REGION Network 15: Interface Signals 10 BK8
   // Call the interface signals bool blocks
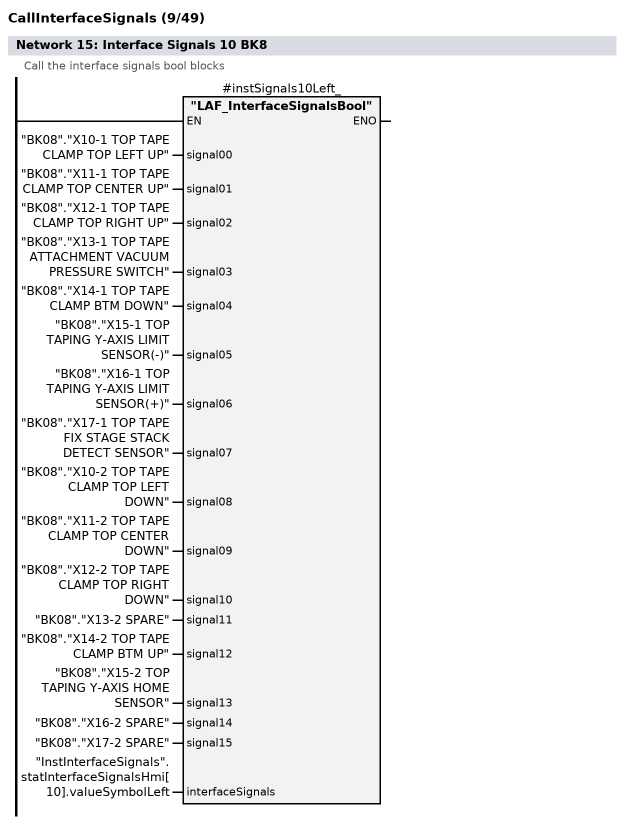
   RUNG wire#powerrail
      #instSignals10Left_(signal00 := "BK08"."X10-1 TOP TAPE CLAMP TOP LEFT UP", signal01 := "BK08"."X11-1 TOP TAPE CLAMP TOP CENTER UP", signal02 := "BK08"."X12-1 TOP TAPE CLAMP TOP RIGHT UP", signal03 := "BK08"."X13-1 TOP TAPE ATTACHMENT VACUUM PRESSURE SWITCH", signal04 := "BK08"."X14-1 TOP TAPE CLAMP BTM DOWN", signal05 := "BK08"."X15-1 TOP TAPING Y-AXIS LIMIT SENSOR(-)", signal06 := "BK08"."X16-1 TOP TAPING Y-AXIS LIMIT SENSOR(+)", signal07 := "BK08"."X17-1 TOP TAPE FIX STAGE STACK DETECT SENSOR", signal08 := "BK08"."X10-2 TOP TAPE CLAMP TOP LEFT DOWN", signal09 := "BK08"."X11-2 TOP TAPE CLAMP TOP CENTER DOWN", signal10 := "BK08"."X12-2 TOP TAPE CLAMP TOP RIGHT DOWN", signal11 := "BK08"."X13-2 SPARE", signal12 := "BK08"."X14-2 TOP TAPE CLAMP BTM UP", signal13 := "BK08"."X15-2 TOP TAPING Y-AXIS HOME SENSOR", signal14 := "BK08"."X16-2 SPARE", signal15 := "BK08"."X17-2 SPARE", interfaceSignals := "InstInterfaceSignals".statInterfaceSignalsHmi[10].valueSymbolLeft)
   END_RUNG
   // the same network as SCL:
   #instSignals10Left_(signal00 := "BK08"."X10-1 TOP TAPE CLAMP TOP LEFT UP",   // "LAF_InterfaceSignalsBool"
                       signal01 := "BK08"."X11-1 TOP TAPE CLAMP TOP CENTER UP",
                       signal02 := "BK08"."X12-1 TOP TAPE CLAMP TOP RIGHT UP",
                       signal03 := "BK08"."X13-1 TOP TAPE ATTACHMENT VACUUM PRESSURE SWITCH",
                       signal04 := "BK08"."X14-1 TOP TAPE CLAMP BTM DOWN",
                       signal05 := "BK08"."X15-1 TOP TAPING Y-AXIS LIMIT SENSOR(-)",
                       signal06 := "BK08"."X16-1 TOP TAPING Y-AXIS LIMIT SENSOR(+)",
                       signal07 := "BK08"."X17-1 TOP TAPE FIX STAGE STACK DETECT SENSOR",
                       signal08 := "BK08"."X10-2 TOP TAPE CLAMP TOP LEFT DOWN",
                       signal09 := "BK08"."X11-2 TOP TAPE CLAMP TOP CENTER DOWN",
                       signal10 := "BK08"."X12-2 TOP TAPE CLAMP TOP RIGHT DOWN",
                       signal11 := "BK08"."X13-2 SPARE",
                       signal12 := "BK08"."X14-2 TOP TAPE CLAMP BTM UP",
                       signal13 := "BK08"."X15-2 TOP TAPING Y-AXIS HOME SENSOR",
                       signal14 := "BK08"."X16-2 SPARE",
                       signal15 := "BK08"."X17-2 SPARE",
                       interfaceSignals := "InstInterfaceSignals".statInterfaceSignalsHmi[10].valueSymbolLeft);
END_REGION

REGION Network 16: Interface Signals 11 BK9
   // Call the interface signals bool blocks
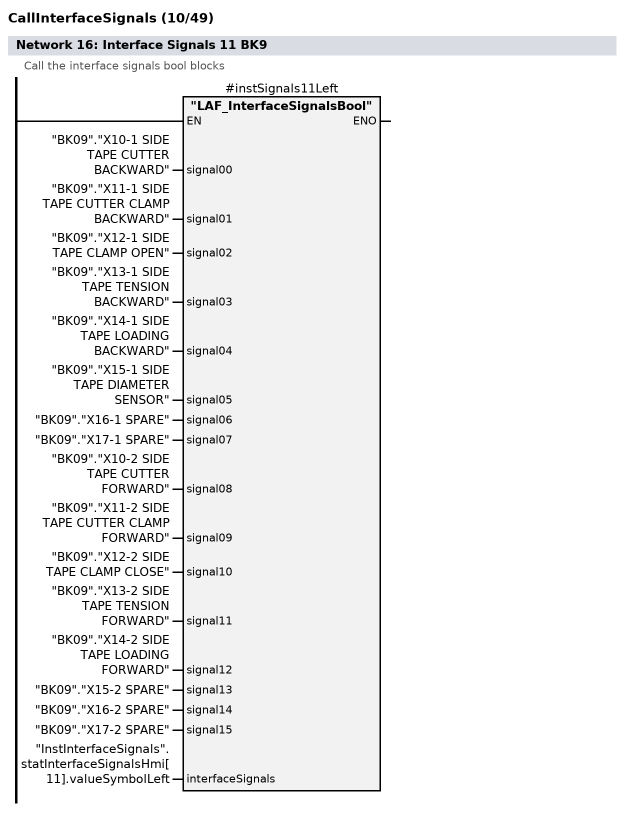
   RUNG wire#powerrail
      #instSignals11Left(signal00 := "BK09"."X10-1 SIDE TAPE CUTTER BACKWARD", signal01 := "BK09"."X11-1 SIDE TAPE CUTTER CLAMP BACKWARD", signal02 := "BK09"."X12-1 SIDE TAPE CLAMP OPEN", signal03 := "BK09"."X13-1 SIDE TAPE TENSION BACKWARD", signal04 := "BK09"."X14-1 SIDE TAPE LOADING BACKWARD", signal05 := "BK09"."X15-1 SIDE TAPE DIAMETER SENSOR", signal06 := "BK09"."X16-1 SPARE", signal07 := "BK09"."X17-1 SPARE", signal08 := "BK09"."X10-2 SIDE TAPE CUTTER FORWARD", signal09 := "BK09"."X11-2 SIDE TAPE CUTTER CLAMP FORWARD", signal10 := "BK09"."X12-2 SIDE TAPE CLAMP CLOSE", signal11 := "BK09"."X13-2 SIDE TAPE TENSION FORWARD", signal12 := "BK09"."X14-2 SIDE TAPE LOADING FORWARD", signal13 := "BK09"."X15-2 SPARE", signal14 := "BK09"."X16-2 SPARE", signal15 := "BK09"."X17-2 SPARE", interfaceSignals := "InstInterfaceSignals".statInterfaceSignalsHmi[11].valueSymbolLeft)
   END_RUNG
   // the same network as SCL:
   #instSignals11Left(signal00 := "BK09"."X10-1 SIDE TAPE CUTTER BACKWARD",   // "LAF_InterfaceSignalsBool"
                      signal01 := "BK09"."X11-1 SIDE TAPE CUTTER CLAMP BACKWARD",
                      signal02 := "BK09"."X12-1 SIDE TAPE CLAMP OPEN",
                      signal03 := "BK09"."X13-1 SIDE TAPE TENSION BACKWARD",
                      signal04 := "BK09"."X14-1 SIDE TAPE LOADING BACKWARD",
                      signal05 := "BK09"."X15-1 SIDE TAPE DIAMETER SENSOR",
                      signal06 := "BK09"."X16-1 SPARE",
                      signal07 := "BK09"."X17-1 SPARE",
                      signal08 := "BK09"."X10-2 SIDE TAPE CUTTER FORWARD",
                      signal09 := "BK09"."X11-2 SIDE TAPE CUTTER CLAMP FORWARD",
                      signal10 := "BK09"."X12-2 SIDE TAPE CLAMP CLOSE",
                      signal11 := "BK09"."X13-2 SIDE TAPE TENSION FORWARD",
                      signal12 := "BK09"."X14-2 SIDE TAPE LOADING FORWARD",
                      signal13 := "BK09"."X15-2 SPARE",
                      signal14 := "BK09"."X16-2 SPARE",
                      signal15 := "BK09"."X17-2 SPARE",
                      interfaceSignals := "InstInterfaceSignals".statInterfaceSignalsHmi[11].valueSymbolLeft);
END_REGION

REGION Network 17: Interface Signals 12 BK10
   // Call the interface signals bool blocks
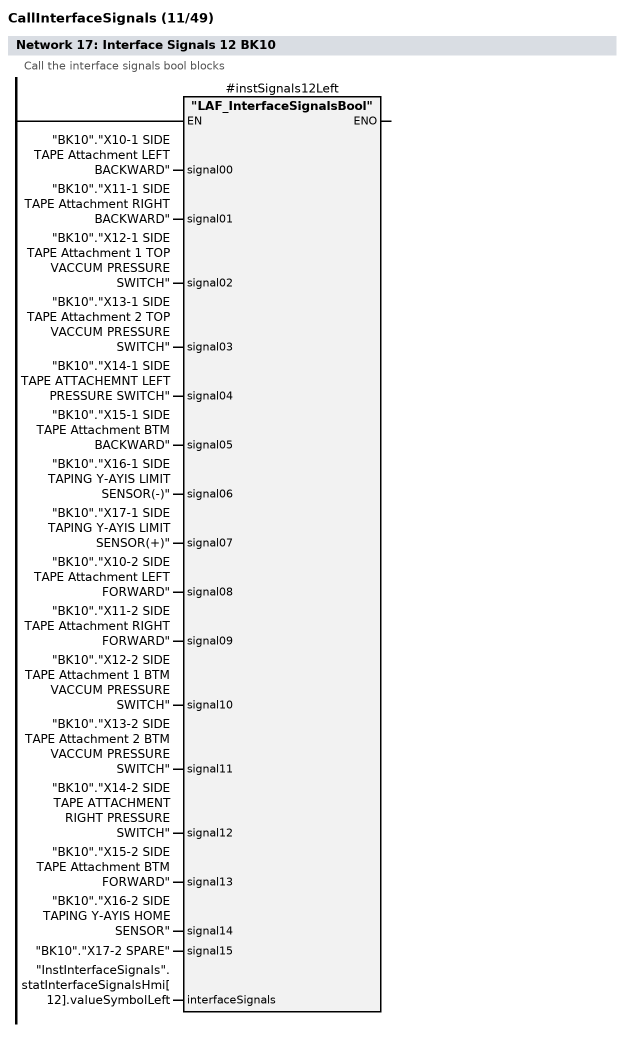
   RUNG wire#powerrail
      #instSignals12Left(signal00 := "BK10"."X10-1 SIDE TAPE Attachment LEFT BACKWARD", signal01 := "BK10"."X11-1 SIDE TAPE Attachment RIGHT BACKWARD", signal02 := "BK10"."X12-1 SIDE TAPE Attachment 1 TOP VACCUM PRESSURE SWITCH", signal03 := "BK10"."X13-1 SIDE TAPE Attachment 2 TOP VACCUM PRESSURE SWITCH", signal04 := "BK10"."X14-1 SIDE TAPE ATTACHEMNT LEFT PRESSURE SWITCH", signal05 := "BK10"."X15-1 SIDE TAPE Attachment BTM BACKWARD", signal06 := "BK10"."X16-1 SIDE TAPING Y-AYIS LIMIT SENSOR(-)", signal07 := "BK10"."X17-1 SIDE TAPING Y-AYIS LIMIT SENSOR(+)", signal08 := "BK10"."X10-2 SIDE TAPE Attachment LEFT FORWARD", signal09 := "BK10"."X11-2 SIDE TAPE Attachment RIGHT FORWARD", signal10 := "BK10"."X12-2 SIDE TAPE Attachment 1 BTM VACCUM PRESSURE SWITCH", signal11 := "BK10"."X13-2 SIDE TAPE Attachment 2 BTM VACCUM PRESSURE SWITCH", signal12 := "BK10"."X14-2 SIDE TAPE ATTACHMENT RIGHT PRESSURE SWITCH", signal13 := "BK10"."X15-2 SIDE TAPE Attachment BTM FORWARD", signal14 := "BK10"."X16-2 SIDE TAPING Y-AYIS HOME SENSOR", signal15 := "BK10"."X17-2 SPARE", interfaceSignals := "InstInterfaceSignals".statInterfaceSignalsHmi[12].valueSymbolLeft)
   END_RUNG
   // the same network as SCL:
   #instSignals12Left(signal00 := "BK10"."X10-1 SIDE TAPE Attachment LEFT BACKWARD",   // "LAF_InterfaceSignalsBool"
                      signal01 := "BK10"."X11-1 SIDE TAPE Attachment RIGHT BACKWARD",
                      signal02 := "BK10"."X12-1 SIDE TAPE Attachment 1 TOP VACCUM PRESSURE SWITCH",
                      signal03 := "BK10"."X13-1 SIDE TAPE Attachment 2 TOP VACCUM PRESSURE SWITCH",
                      signal04 := "BK10"."X14-1 SIDE TAPE ATTACHEMNT LEFT PRESSURE SWITCH",
                      signal05 := "BK10"."X15-1 SIDE TAPE Attachment BTM BACKWARD",
                      signal06 := "BK10"."X16-1 SIDE TAPING Y-AYIS LIMIT SENSOR(-)",
                      signal07 := "BK10"."X17-1 SIDE TAPING Y-AYIS LIMIT SENSOR(+)",
                      signal08 := "BK10"."X10-2 SIDE TAPE Attachment LEFT FORWARD",
                      signal09 := "BK10"."X11-2 SIDE TAPE Attachment RIGHT FORWARD",
                      signal10 := "BK10"."X12-2 SIDE TAPE Attachment 1 BTM VACCUM PRESSURE SWITCH",
                      signal11 := "BK10"."X13-2 SIDE TAPE Attachment 2 BTM VACCUM PRESSURE SWITCH",
                      signal12 := "BK10"."X14-2 SIDE TAPE ATTACHMENT RIGHT PRESSURE SWITCH",
                      signal13 := "BK10"."X15-2 SIDE TAPE Attachment BTM FORWARD",
                      signal14 := "BK10"."X16-2 SIDE TAPING Y-AYIS HOME SENSOR",
                      signal15 := "BK10"."X17-2 SPARE",
                      interfaceSignals := "InstInterfaceSignals".statInterfaceSignalsHmi[12].valueSymbolLeft);
END_REGION

REGION Network 18: Interface Signals 13 BK11
   // Call the interface signals bool blocks
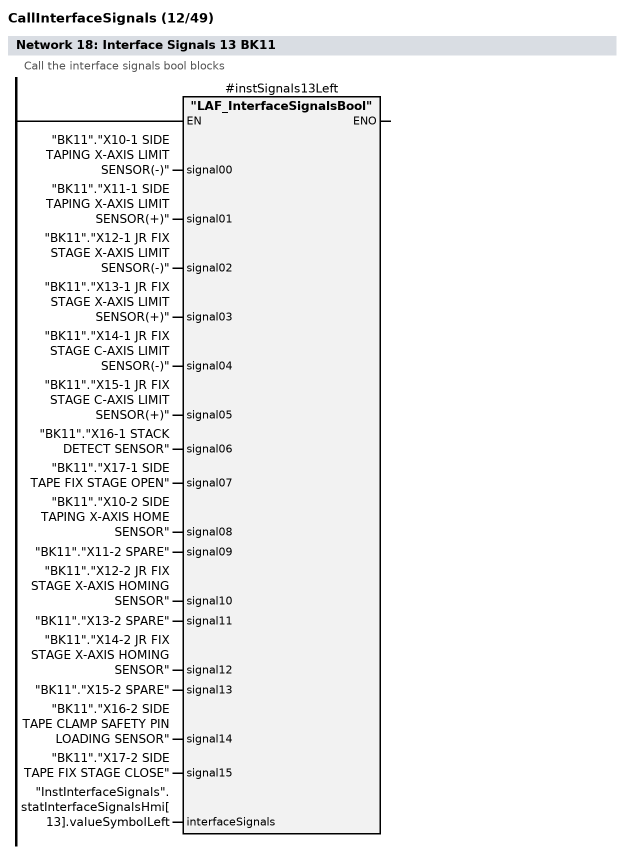
   RUNG wire#powerrail
      #instSignals13Left(signal00 := "BK11"."X10-1 SIDE TAPING X-AXIS LIMIT SENSOR(-)", signal01 := "BK11"."X11-1 SIDE TAPING X-AXIS LIMIT SENSOR(+)", signal02 := "BK11"."X12-1 JR FIX STAGE X-AXIS LIMIT SENSOR(-)", signal03 := "BK11"."X13-1 JR FIX STAGE X-AXIS LIMIT SENSOR(+)", signal04 := "BK11"."X14-1 JR FIX STAGE C-AXIS LIMIT SENSOR(-)", signal05 := "BK11"."X15-1 JR FIX STAGE C-AXIS LIMIT SENSOR(+)", signal06 := "BK11"."X16-1 STACK DETECT SENSOR", signal07 := "BK11"."X17-1 SIDE TAPE FIX STAGE OPEN", signal08 := "BK11"."X10-2 SIDE TAPING X-AXIS HOME SENSOR", signal09 := "BK11"."X11-2 SPARE", signal10 := "BK11"."X12-2 JR FIX STAGE X-AXIS HOMING SENSOR", signal11 := "BK11"."X13-2 SPARE", signal12 := "BK11"."X14-2 JR FIX STAGE X-AXIS HOMING SENSOR", signal13 := "BK11"."X15-2 SPARE", signal14 := "BK11"."X16-2 SIDE TAPE CLAMP SAFETY PIN LOADING SENSOR", signal15 := "BK11"."X17-2 SIDE TAPE FIX STAGE CLOSE", interfaceSignals := "InstInterfaceSignals".statInterfaceSignalsHmi[13].valueSymbolLeft)
   END_RUNG
   // the same network as SCL:
   #instSignals13Left(signal00 := "BK11"."X10-1 SIDE TAPING X-AXIS LIMIT SENSOR(-)",   // "LAF_InterfaceSignalsBool"
                      signal01 := "BK11"."X11-1 SIDE TAPING X-AXIS LIMIT SENSOR(+)",
                      signal02 := "BK11"."X12-1 JR FIX STAGE X-AXIS LIMIT SENSOR(-)",
                      signal03 := "BK11"."X13-1 JR FIX STAGE X-AXIS LIMIT SENSOR(+)",
                      signal04 := "BK11"."X14-1 JR FIX STAGE C-AXIS LIMIT SENSOR(-)",
                      signal05 := "BK11"."X15-1 JR FIX STAGE C-AXIS LIMIT SENSOR(+)",
                      signal06 := "BK11"."X16-1 STACK DETECT SENSOR",
                      signal07 := "BK11"."X17-1 SIDE TAPE FIX STAGE OPEN",
                      signal08 := "BK11"."X10-2 SIDE TAPING X-AXIS HOME SENSOR",
                      signal09 := "BK11"."X11-2 SPARE",
                      signal10 := "BK11"."X12-2 JR FIX STAGE X-AXIS HOMING SENSOR",
                      signal11 := "BK11"."X13-2 SPARE",
                      signal12 := "BK11"."X14-2 JR FIX STAGE X-AXIS HOMING SENSOR",
                      signal13 := "BK11"."X15-2 SPARE",
                      signal14 := "BK11"."X16-2 SIDE TAPE CLAMP SAFETY PIN LOADING SENSOR",
                      signal15 := "BK11"."X17-2 SIDE TAPE FIX STAGE CLOSE",
                      interfaceSignals := "InstInterfaceSignals".statInterfaceSignalsHmi[13].valueSymbolLeft);
END_REGION

REGION Network 19: Interface Signals 14 BK12
   // Call the interface signals bool blocks
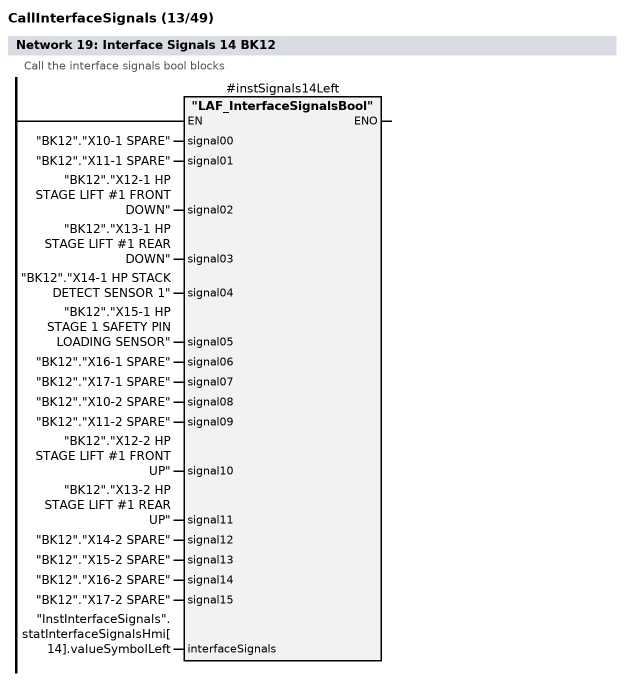
   RUNG wire#powerrail
      #instSignals14Left(signal00 := "BK12"."X10-1 SPARE", signal01 := "BK12"."X11-1 SPARE", signal02 := "BK12"."X12-1 HP STAGE LIFT #1 FRONT DOWN", signal03 := "BK12"."X13-1 HP STAGE LIFT #1 REAR DOWN", signal04 := "BK12"."X14-1 HP STACK DETECT SENSOR 1", signal05 := "BK12"."X15-1 HP STAGE 1 SAFETY PIN LOADING SENSOR", signal06 := "BK12"."X16-1 SPARE", signal07 := "BK12"."X17-1 SPARE", signal08 := "BK12"."X10-2 SPARE", signal09 := "BK12"."X11-2 SPARE", signal10 := "BK12"."X12-2 HP STAGE LIFT #1 FRONT UP", signal11 := "BK12"."X13-2 HP STAGE LIFT #1 REAR UP", signal12 := "BK12"."X14-2 SPARE", signal13 := "BK12"."X15-2 SPARE", signal14 := "BK12"."X16-2 SPARE", signal15 := "BK12"."X17-2 SPARE", interfaceSignals := "InstInterfaceSignals".statInterfaceSignalsHmi[14].valueSymbolLeft)
   END_RUNG
   // the same network as SCL:
   #instSignals14Left(signal00 := "BK12"."X10-1 SPARE",   // "LAF_InterfaceSignalsBool"
                      signal01 := "BK12"."X11-1 SPARE",
                      signal02 := "BK12"."X12-1 HP STAGE LIFT #1 FRONT DOWN",
                      signal03 := "BK12"."X13-1 HP STAGE LIFT #1 REAR DOWN",
                      signal04 := "BK12"."X14-1 HP STACK DETECT SENSOR 1",
                      signal05 := "BK12"."X15-1 HP STAGE 1 SAFETY PIN LOADING SENSOR",
                      signal06 := "BK12"."X16-1 SPARE",
                      signal07 := "BK12"."X17-1 SPARE",
                      signal08 := "BK12"."X10-2 SPARE",
                      signal09 := "BK12"."X11-2 SPARE",
                      signal10 := "BK12"."X12-2 HP STAGE LIFT #1 FRONT UP",
                      signal11 := "BK12"."X13-2 HP STAGE LIFT #1 REAR UP",
                      signal12 := "BK12"."X14-2 SPARE",
                      signal13 := "BK12"."X15-2 SPARE",
                      signal14 := "BK12"."X16-2 SPARE",
                      signal15 := "BK12"."X17-2 SPARE",
                      interfaceSignals := "InstInterfaceSignals".statInterfaceSignalsHmi[14].valueSymbolLeft);
END_REGION

REGION Network 20: Interface Signals 15 BK13
   // Call the interface signals bool blocks
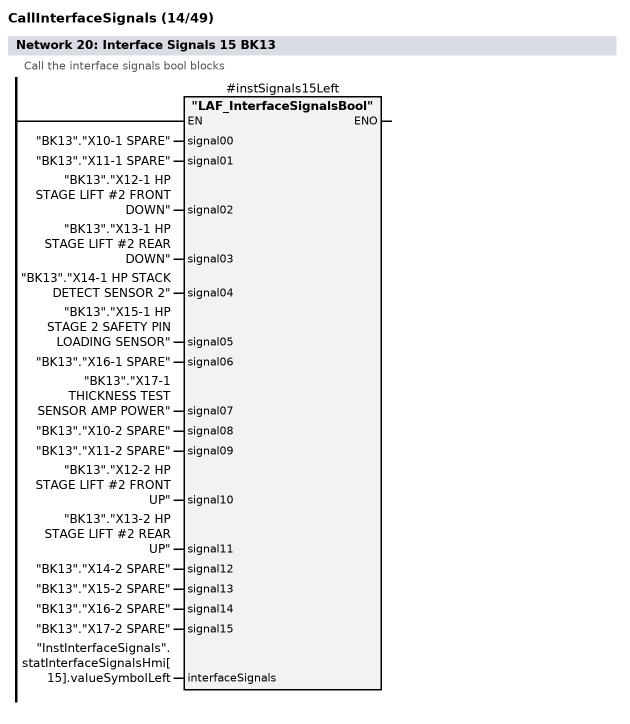
   RUNG wire#powerrail
      #instSignals15Left(signal00 := "BK13"."X10-1 SPARE", signal01 := "BK13"."X11-1 SPARE", signal02 := "BK13"."X12-1 HP STAGE LIFT #2 FRONT DOWN", signal03 := "BK13"."X13-1 HP STAGE LIFT #2 REAR DOWN", signal04 := "BK13"."X14-1 HP STACK DETECT SENSOR 2", signal05 := "BK13"."X15-1 HP STAGE 2 SAFETY PIN LOADING SENSOR", signal06 := "BK13"."X16-1 SPARE", signal07 := "BK13"."X17-1 THICKNESS TEST SENSOR AMP POWER", signal08 := "BK13"."X10-2 SPARE", signal09 := "BK13"."X11-2 SPARE", signal10 := "BK13"."X12-2 HP STAGE LIFT #2 FRONT UP", signal11 := "BK13"."X13-2 HP STAGE LIFT #2 REAR UP", signal12 := "BK13"."X14-2 SPARE", signal13 := "BK13"."X15-2 SPARE", signal14 := "BK13"."X16-2 SPARE", signal15 := "BK13"."X17-2 SPARE", interfaceSignals := "InstInterfaceSignals".statInterfaceSignalsHmi[15].valueSymbolLeft)
   END_RUNG
   // the same network as SCL:
   #instSignals15Left(signal00 := "BK13"."X10-1 SPARE",   // "LAF_InterfaceSignalsBool"
                      signal01 := "BK13"."X11-1 SPARE",
                      signal02 := "BK13"."X12-1 HP STAGE LIFT #2 FRONT DOWN",
                      signal03 := "BK13"."X13-1 HP STAGE LIFT #2 REAR DOWN",
                      signal04 := "BK13"."X14-1 HP STACK DETECT SENSOR 2",
                      signal05 := "BK13"."X15-1 HP STAGE 2 SAFETY PIN LOADING SENSOR",
                      signal06 := "BK13"."X16-1 SPARE",
                      signal07 := "BK13"."X17-1 THICKNESS TEST SENSOR AMP POWER",
                      signal08 := "BK13"."X10-2 SPARE",
                      signal09 := "BK13"."X11-2 SPARE",
                      signal10 := "BK13"."X12-2 HP STAGE LIFT #2 FRONT UP",
                      signal11 := "BK13"."X13-2 HP STAGE LIFT #2 REAR UP",
                      signal12 := "BK13"."X14-2 SPARE",
                      signal13 := "BK13"."X15-2 SPARE",
                      signal14 := "BK13"."X16-2 SPARE",
                      signal15 := "BK13"."X17-2 SPARE",
                      interfaceSignals := "InstInterfaceSignals".statInterfaceSignalsHmi[15].valueSymbolLeft);
END_REGION

REGION Network 21: Interface Signals 16 BK14
   // Call the interface signals bool blocks
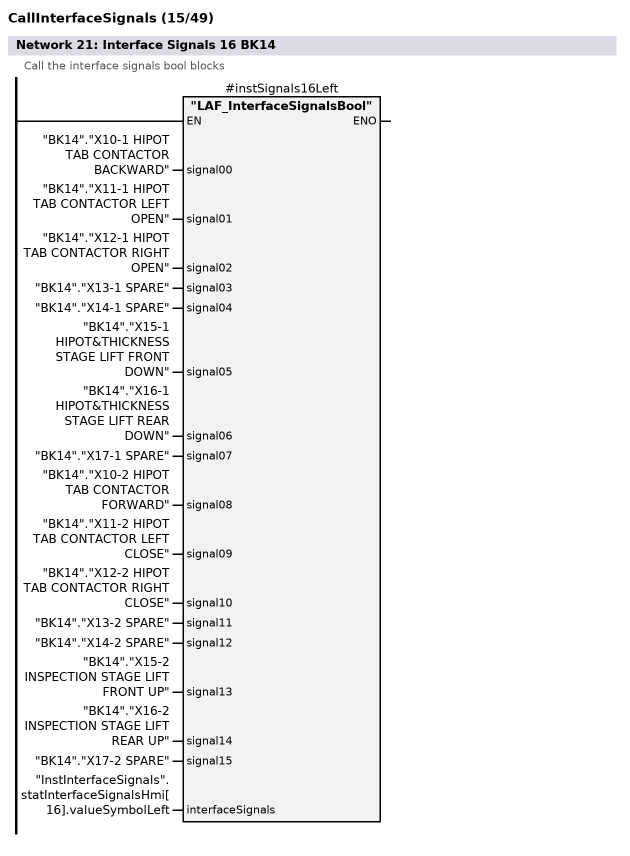
   RUNG wire#powerrail
      #instSignals16Left(signal00 := "BK14"."X10-1 HIPOT TAB CONTACTOR BACKWARD", signal01 := "BK14"."X11-1 HIPOT TAB CONTACTOR LEFT OPEN", signal02 := "BK14"."X12-1 HIPOT TAB CONTACTOR RIGHT OPEN", signal03 := "BK14"."X13-1 SPARE", signal04 := "BK14"."X14-1 SPARE", signal05 := "BK14"."X15-1 HIPOT&THICKNESS STAGE LIFT FRONT DOWN", signal06 := "BK14"."X16-1 HIPOT&THICKNESS STAGE LIFT REAR DOWN", signal07 := "BK14"."X17-1 SPARE", signal08 := "BK14"."X10-2 HIPOT TAB CONTACTOR FORWARD", signal09 := "BK14"."X11-2 HIPOT TAB CONTACTOR LEFT CLOSE", signal10 := "BK14"."X12-2 HIPOT TAB CONTACTOR RIGHT CLOSE", signal11 := "BK14"."X13-2 SPARE", signal12 := "BK14"."X14-2 SPARE", signal13 := "BK14"."X15-2 INSPECTION STAGE LIFT FRONT UP", signal14 := "BK14"."X16-2 INSPECTION STAGE LIFT REAR UP", signal15 := "BK14"."X17-2 SPARE", interfaceSignals := "InstInterfaceSignals".statInterfaceSignalsHmi[16].valueSymbolLeft)
   END_RUNG
   // the same network as SCL:
   #instSignals16Left(signal00 := "BK14"."X10-1 HIPOT TAB CONTACTOR BACKWARD",   // "LAF_InterfaceSignalsBool"
                      signal01 := "BK14"."X11-1 HIPOT TAB CONTACTOR LEFT OPEN",
                      signal02 := "BK14"."X12-1 HIPOT TAB CONTACTOR RIGHT OPEN",
                      signal03 := "BK14"."X13-1 SPARE",
                      signal04 := "BK14"."X14-1 SPARE",
                      signal05 := "BK14"."X15-1 HIPOT&THICKNESS STAGE LIFT FRONT DOWN",
                      signal06 := "BK14"."X16-1 HIPOT&THICKNESS STAGE LIFT REAR DOWN",
                      signal07 := "BK14"."X17-1 SPARE",
                      signal08 := "BK14"."X10-2 HIPOT TAB CONTACTOR FORWARD",
                      signal09 := "BK14"."X11-2 HIPOT TAB CONTACTOR LEFT CLOSE",
                      signal10 := "BK14"."X12-2 HIPOT TAB CONTACTOR RIGHT CLOSE",
                      signal11 := "BK14"."X13-2 SPARE",
                      signal12 := "BK14"."X14-2 SPARE",
                      signal13 := "BK14"."X15-2 INSPECTION STAGE LIFT FRONT UP",
                      signal14 := "BK14"."X16-2 INSPECTION STAGE LIFT REAR UP",
                      signal15 := "BK14"."X17-2 SPARE",
                      interfaceSignals := "InstInterfaceSignals".statInterfaceSignalsHmi[16].valueSymbolLeft);
END_REGION

REGION Network 22: Interface Signals 17 BK15
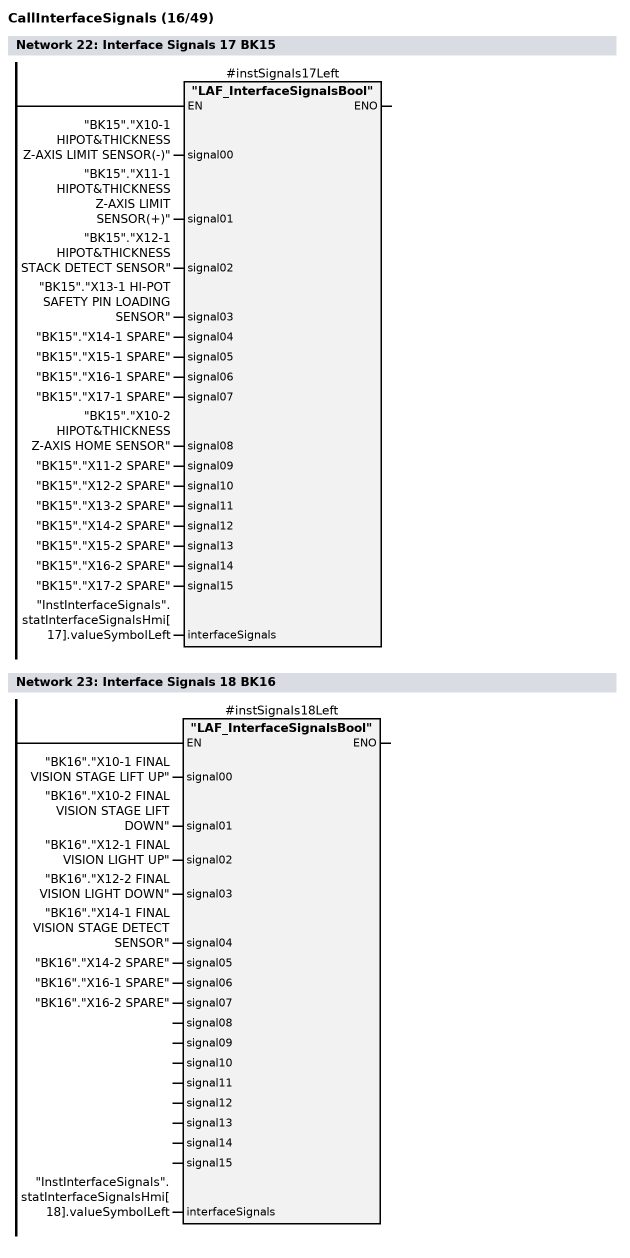
   RUNG wire#powerrail
      #instSignals17Left(signal00 := "BK15"."X10-1 HIPOT&THICKNESS Z-AXIS LIMIT SENSOR(-)", signal01 := "BK15"."X11-1 HIPOT&THICKNESS Z-AXIS LIMIT SENSOR(+)", signal02 := "BK15"."X12-1 HIPOT&THICKNESS STACK DETECT SENSOR", signal03 := "BK15"."X13-1 HI-POT SAFETY PIN LOADING SENSOR", signal04 := "BK15"."X14-1 SPARE", signal05 := "BK15"."X15-1 SPARE", signal06 := "BK15"."X16-1 SPARE", signal07 := "BK15"."X17-1 SPARE", signal08 := "BK15"."X10-2 HIPOT&THICKNESS Z-AXIS HOME SENSOR", signal09 := "BK15"."X11-2 SPARE", signal10 := "BK15"."X12-2 SPARE", signal11 := "BK15"."X13-2 SPARE", signal12 := "BK15"."X14-2 SPARE", signal13 := "BK15"."X15-2 SPARE", signal14 := "BK15"."X16-2 SPARE", signal15 := "BK15"."X17-2 SPARE", interfaceSignals := "InstInterfaceSignals".statInterfaceSignalsHmi[17].valueSymbolLeft)
   END_RUNG
   // the same network as SCL:
   #instSignals17Left(signal00 := "BK15"."X10-1 HIPOT&THICKNESS Z-AXIS LIMIT SENSOR(-)",   // "LAF_InterfaceSignalsBool"
                      signal01 := "BK15"."X11-1 HIPOT&THICKNESS Z-AXIS LIMIT SENSOR(+)",
                      signal02 := "BK15"."X12-1 HIPOT&THICKNESS STACK DETECT SENSOR",
                      signal03 := "BK15"."X13-1 HI-POT SAFETY PIN LOADING SENSOR",
                      signal04 := "BK15"."X14-1 SPARE",
                      signal05 := "BK15"."X15-1 SPARE",
                      signal06 := "BK15"."X16-1 SPARE",
                      signal07 := "BK15"."X17-1 SPARE",
                      signal08 := "BK15"."X10-2 HIPOT&THICKNESS Z-AXIS HOME SENSOR",
                      signal09 := "BK15"."X11-2 SPARE",
                      signal10 := "BK15"."X12-2 SPARE",
                      signal11 := "BK15"."X13-2 SPARE",
                      signal12 := "BK15"."X14-2 SPARE",
                      signal13 := "BK15"."X15-2 SPARE",
                      signal14 := "BK15"."X16-2 SPARE",
                      signal15 := "BK15"."X17-2 SPARE",
                      interfaceSignals := "InstInterfaceSignals".statInterfaceSignalsHmi[17].valueSymbolLeft);
END_REGION

REGION Network 23: Interface Signals 18 BK16
   RUNG wire#powerrail
      #instSignals18Left(signal00 := "BK16"."X10-1 FINAL VISION STAGE LIFT UP", signal01 := "BK16"."X10-2 FINAL VISION STAGE LIFT DOWN", signal02 := "BK16"."X12-1 FINAL VISION LIGHT UP", signal03 := "BK16"."X12-2 FINAL VISION LIGHT DOWN", signal04 := "BK16"."X14-1 FINAL VISION STAGE DETECT SENSOR", signal05 := "BK16"."X14-2 SPARE", signal06 := "BK16"."X16-1 SPARE", signal07 := "BK16"."X16-2 SPARE", signal08 :=, signal09 :=, signal10 :=, signal11 :=, signal12 :=, signal13 :=, signal14 :=, signal15 :=, interfaceSignals := "InstInterfaceSignals".statInterfaceSignalsHmi[18].valueSymbolLeft)
   END_RUNG
   // the same network as SCL:
   #instSignals18Left(signal00 := "BK16"."X10-1 FINAL VISION STAGE LIFT UP",   // "LAF_InterfaceSignalsBool"
                      signal01 := "BK16"."X10-2 FINAL VISION STAGE LIFT DOWN",
                      signal02 := "BK16"."X12-1 FINAL VISION LIGHT UP",
                      signal03 := "BK16"."X12-2 FINAL VISION LIGHT DOWN",
                      signal04 := "BK16"."X14-1 FINAL VISION STAGE DETECT SENSOR",
                      signal05 := "BK16"."X14-2 SPARE",
                      signal06 := "BK16"."X16-1 SPARE",
                      signal07 := "BK16"."X16-2 SPARE",
                      interfaceSignals := "InstInterfaceSignals".statInterfaceSignalsHmi[18].valueSymbolLeft);
END_REGION

REGION Network 24: Interface Signals 19 BK17
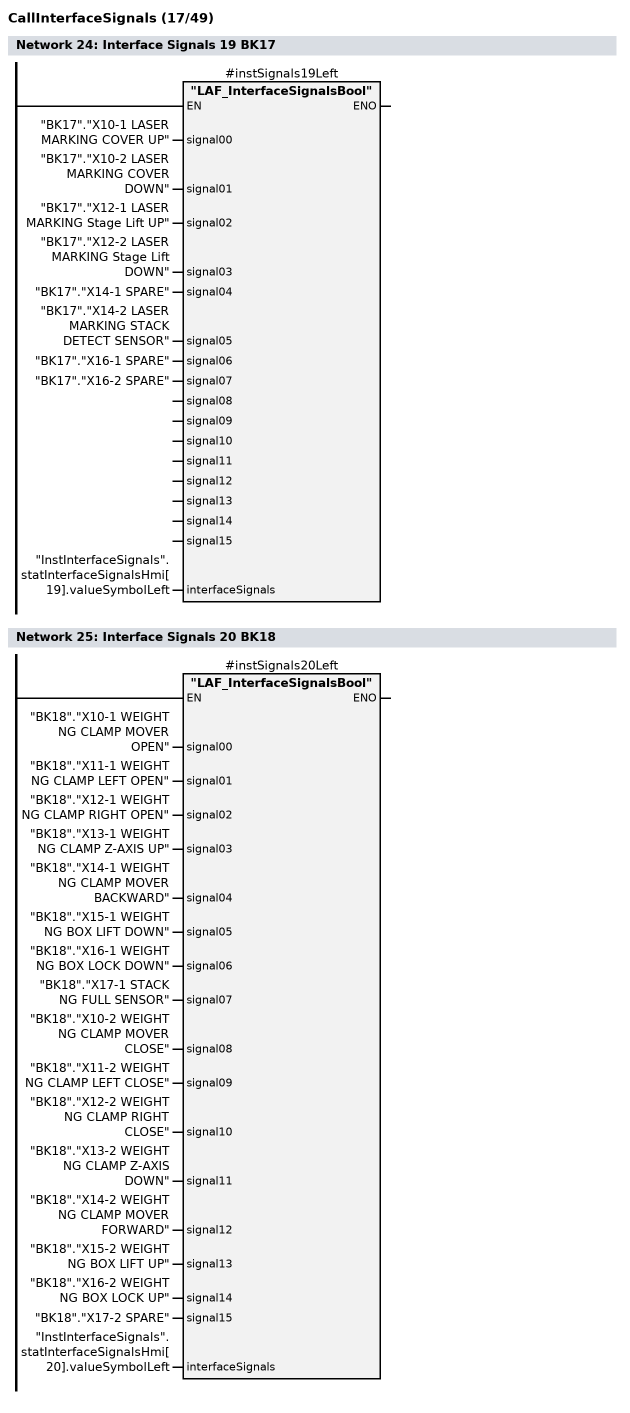
   RUNG wire#powerrail
      #instSignals19Left(signal00 := "BK17"."X10-1 LASER MARKING COVER UP", signal01 := "BK17"."X10-2 LASER MARKING COVER DOWN", signal02 := "BK17"."X12-1 LASER MARKING Stage Lift UP", signal03 := "BK17"."X12-2 LASER MARKING Stage Lift DOWN", signal04 := "BK17"."X14-1 SPARE", signal05 := "BK17"."X14-2 LASER MARKING STACK DETECT SENSOR", signal06 := "BK17"."X16-1 SPARE", signal07 := "BK17"."X16-2 SPARE", signal08 :=, signal09 :=, signal10 :=, signal11 :=, signal12 :=, signal13 :=, signal14 :=, signal15 :=, interfaceSignals := "InstInterfaceSignals".statInterfaceSignalsHmi[19].valueSymbolLeft)
   END_RUNG
   // the same network as SCL:
   #instSignals19Left(signal00 := "BK17"."X10-1 LASER MARKING COVER UP",   // "LAF_InterfaceSignalsBool"
                      signal01 := "BK17"."X10-2 LASER MARKING COVER DOWN",
                      signal02 := "BK17"."X12-1 LASER MARKING Stage Lift UP",
                      signal03 := "BK17"."X12-2 LASER MARKING Stage Lift DOWN",
                      signal04 := "BK17"."X14-1 SPARE",
                      signal05 := "BK17"."X14-2 LASER MARKING STACK DETECT SENSOR",
                      signal06 := "BK17"."X16-1 SPARE",
                      signal07 := "BK17"."X16-2 SPARE",
                      interfaceSignals := "InstInterfaceSignals".statInterfaceSignalsHmi[19].valueSymbolLeft);
END_REGION

REGION Network 25: Interface Signals 20 BK18
   RUNG wire#powerrail
      #instSignals20Left(signal00 := "BK18"."X10-1 WEIGHT NG CLAMP MOVER OPEN", signal01 := "BK18"."X11-1 WEIGHT NG CLAMP LEFT OPEN", signal02 := "BK18"."X12-1 WEIGHT NG CLAMP RIGHT OPEN", signal03 := "BK18"."X13-1 WEIGHT NG CLAMP Z-AXIS UP", signal04 := "BK18"."X14-1 WEIGHT NG CLAMP MOVER BACKWARD", signal05 := "BK18"."X15-1 WEIGHT NG BOX LIFT DOWN", signal06 := "BK18"."X16-1 WEIGHT NG BOX LOCK DOWN", signal07 := "BK18"."X17-1 STACK NG FULL SENSOR", signal08 := "BK18"."X10-2 WEIGHT NG CLAMP MOVER CLOSE", signal09 := "BK18"."X11-2 WEIGHT NG CLAMP LEFT CLOSE", signal10 := "BK18"."X12-2 WEIGHT NG CLAMP RIGHT CLOSE", signal11 := "BK18"."X13-2 WEIGHT NG CLAMP Z-AXIS DOWN", signal12 := "BK18"."X14-2 WEIGHT NG CLAMP MOVER FORWARD", signal13 := "BK18"."X15-2 WEIGHT NG BOX LIFT UP", signal14 := "BK18"."X16-2 WEIGHT NG BOX LOCK UP", signal15 := "BK18"."X17-2 SPARE", interfaceSignals := "InstInterfaceSignals".statInterfaceSignalsHmi[20].valueSymbolLeft)
   END_RUNG
   // the same network as SCL:
   #instSignals20Left(signal00 := "BK18"."X10-1 WEIGHT NG CLAMP MOVER OPEN",   // "LAF_InterfaceSignalsBool"
                      signal01 := "BK18"."X11-1 WEIGHT NG CLAMP LEFT OPEN",
                      signal02 := "BK18"."X12-1 WEIGHT NG CLAMP RIGHT OPEN",
                      signal03 := "BK18"."X13-1 WEIGHT NG CLAMP Z-AXIS UP",
                      signal04 := "BK18"."X14-1 WEIGHT NG CLAMP MOVER BACKWARD",
                      signal05 := "BK18"."X15-1 WEIGHT NG BOX LIFT DOWN",
                      signal06 := "BK18"."X16-1 WEIGHT NG BOX LOCK DOWN",
                      signal07 := "BK18"."X17-1 STACK NG FULL SENSOR",
                      signal08 := "BK18"."X10-2 WEIGHT NG CLAMP MOVER CLOSE",
                      signal09 := "BK18"."X11-2 WEIGHT NG CLAMP LEFT CLOSE",
                      signal10 := "BK18"."X12-2 WEIGHT NG CLAMP RIGHT CLOSE",
                      signal11 := "BK18"."X13-2 WEIGHT NG CLAMP Z-AXIS DOWN",
                      signal12 := "BK18"."X14-2 WEIGHT NG CLAMP MOVER FORWARD",
                      signal13 := "BK18"."X15-2 WEIGHT NG BOX LIFT UP",
                      signal14 := "BK18"."X16-2 WEIGHT NG BOX LOCK UP",
                      signal15 := "BK18"."X17-2 SPARE",
                      interfaceSignals := "InstInterfaceSignals".statInterfaceSignalsHmi[20].valueSymbolLeft);
END_REGION

REGION Network 26: Interface Signals 21 BK19
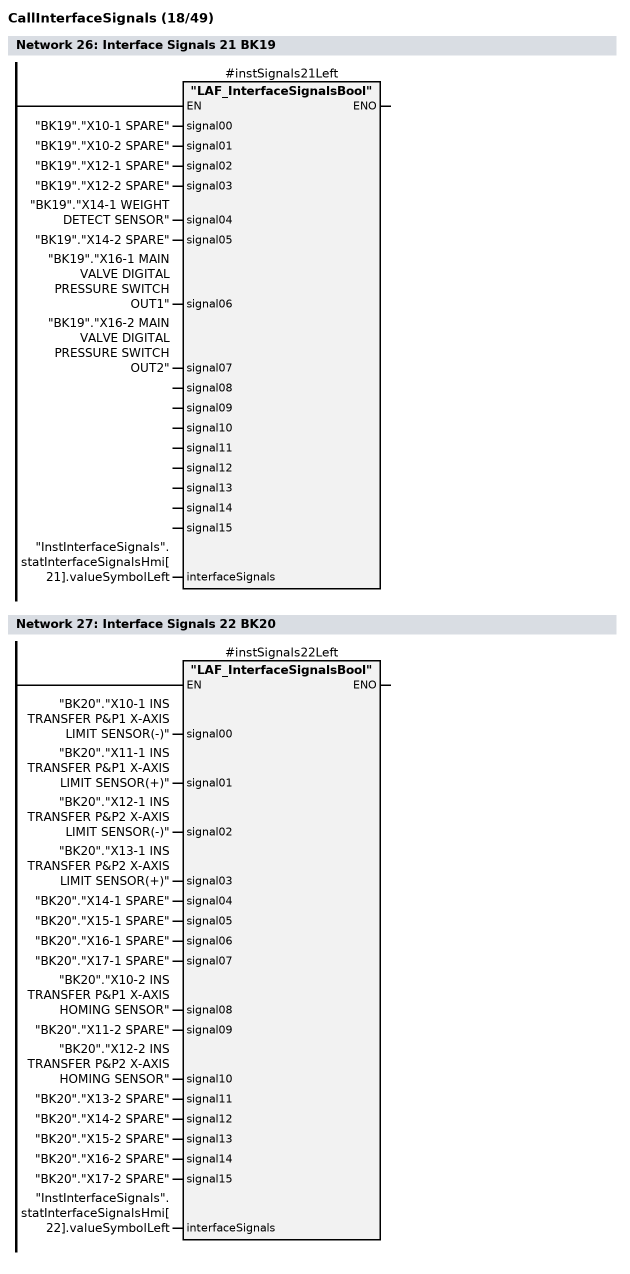
   RUNG wire#powerrail
      #instSignals21Left(signal00 := "BK19"."X10-1 SPARE", signal01 := "BK19"."X10-2 SPARE", signal02 := "BK19"."X12-1 SPARE", signal03 := "BK19"."X12-2 SPARE", signal04 := "BK19"."X14-1 WEIGHT DETECT SENSOR", signal05 := "BK19"."X14-2 SPARE", signal06 := "BK19"."X16-1 MAIN VALVE DIGITAL PRESSURE SWITCH OUT1", signal07 := "BK19"."X16-2 MAIN VALVE DIGITAL PRESSURE SWITCH OUT2", signal08 :=, signal09 :=, signal10 :=, signal11 :=, signal12 :=, signal13 :=, signal14 :=, signal15 :=, interfaceSignals := "InstInterfaceSignals".statInterfaceSignalsHmi[21].valueSymbolLeft)
   END_RUNG
   // the same network as SCL:
   #instSignals21Left(signal00 := "BK19"."X10-1 SPARE",   // "LAF_InterfaceSignalsBool"
                      signal01 := "BK19"."X10-2 SPARE",
                      signal02 := "BK19"."X12-1 SPARE",
                      signal03 := "BK19"."X12-2 SPARE",
                      signal04 := "BK19"."X14-1 WEIGHT DETECT SENSOR",
                      signal05 := "BK19"."X14-2 SPARE",
                      signal06 := "BK19"."X16-1 MAIN VALVE DIGITAL PRESSURE SWITCH OUT1",
                      signal07 := "BK19"."X16-2 MAIN VALVE DIGITAL PRESSURE SWITCH OUT2",
                      interfaceSignals := "InstInterfaceSignals".statInterfaceSignalsHmi[21].valueSymbolLeft);
END_REGION

REGION Network 27: Interface Signals 22 BK20
   RUNG wire#powerrail
      #instSignals22Left(signal00 := "BK20"."X10-1 INS TRANSFER P&P1 X-AXIS LIMIT SENSOR(-)", signal01 := "BK20"."X11-1 INS TRANSFER P&P1 X-AXIS LIMIT SENSOR(+)", signal02 := "BK20"."X12-1 INS TRANSFER P&P2 X-AXIS LIMIT SENSOR(-)", signal03 := "BK20"."X13-1 INS TRANSFER P&P2 X-AXIS LIMIT SENSOR(+)", signal04 := "BK20"."X14-1 SPARE", signal05 := "BK20"."X15-1 SPARE", signal06 := "BK20"."X16-1 SPARE", signal07 := "BK20"."X17-1 SPARE", signal08 := "BK20"."X10-2 INS TRANSFER P&P1 X-AXIS HOMING SENSOR", signal09 := "BK20"."X11-2 SPARE", signal10 := "BK20"."X12-2 INS TRANSFER P&P2 X-AXIS HOMING SENSOR", signal11 := "BK20"."X13-2 SPARE", signal12 := "BK20"."X14-2 SPARE", signal13 := "BK20"."X15-2 SPARE", signal14 := "BK20"."X16-2 SPARE", signal15 := "BK20"."X17-2 SPARE", interfaceSignals := "InstInterfaceSignals".statInterfaceSignalsHmi[22].valueSymbolLeft)
   END_RUNG
   // the same network as SCL:
   #instSignals22Left(signal00 := "BK20"."X10-1 INS TRANSFER P&P1 X-AXIS LIMIT SENSOR(-)",   // "LAF_InterfaceSignalsBool"
                      signal01 := "BK20"."X11-1 INS TRANSFER P&P1 X-AXIS LIMIT SENSOR(+)",
                      signal02 := "BK20"."X12-1 INS TRANSFER P&P2 X-AXIS LIMIT SENSOR(-)",
                      signal03 := "BK20"."X13-1 INS TRANSFER P&P2 X-AXIS LIMIT SENSOR(+)",
                      signal04 := "BK20"."X14-1 SPARE",
                      signal05 := "BK20"."X15-1 SPARE",
                      signal06 := "BK20"."X16-1 SPARE",
                      signal07 := "BK20"."X17-1 SPARE",
                      signal08 := "BK20"."X10-2 INS TRANSFER P&P1 X-AXIS HOMING SENSOR",
                      signal09 := "BK20"."X11-2 SPARE",
                      signal10 := "BK20"."X12-2 INS TRANSFER P&P2 X-AXIS HOMING SENSOR",
                      signal11 := "BK20"."X13-2 SPARE",
                      signal12 := "BK20"."X14-2 SPARE",
                      signal13 := "BK20"."X15-2 SPARE",
                      signal14 := "BK20"."X16-2 SPARE",
                      signal15 := "BK20"."X17-2 SPARE",
                      interfaceSignals := "InstInterfaceSignals".statInterfaceSignalsHmi[22].valueSymbolLeft);
END_REGION

REGION Network 28: Interface Signals 23 BK21
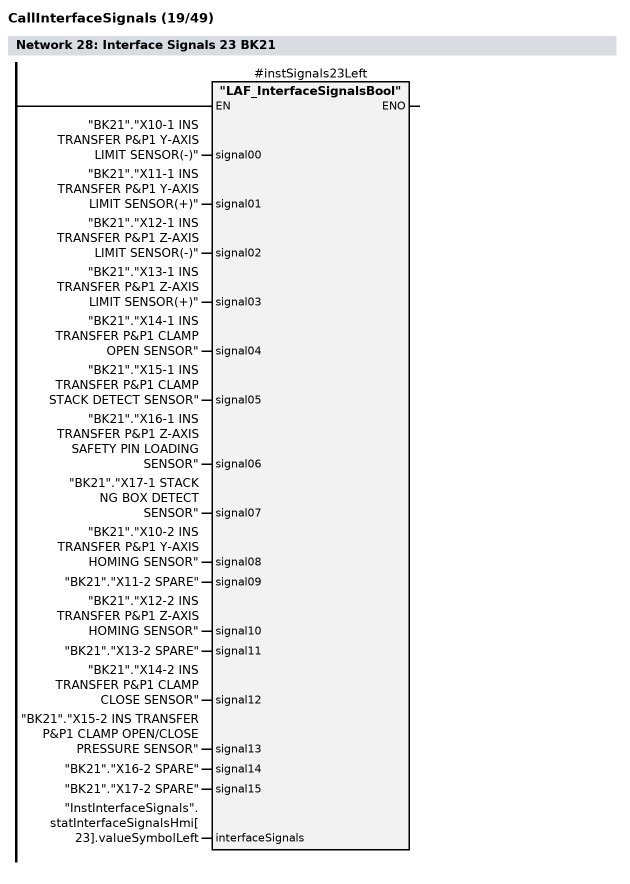
   RUNG wire#powerrail
      #instSignals23Left(signal00 := "BK21"."X10-1 INS TRANSFER P&P1 Y-AXIS LIMIT SENSOR(-)", signal01 := "BK21"."X11-1 INS TRANSFER P&P1 Y-AXIS LIMIT SENSOR(+)", signal02 := "BK21"."X12-1 INS TRANSFER P&P1 Z-AXIS LIMIT SENSOR(-)", signal03 := "BK21"."X13-1 INS TRANSFER P&P1 Z-AXIS LIMIT SENSOR(+)", signal04 := "BK21"."X14-1 INS TRANSFER P&P1 CLAMP OPEN SENSOR", signal05 := "BK21"."X15-1 INS TRANSFER P&P1 CLAMP STACK DETECT SENSOR", signal06 := "BK21"."X16-1 INS TRANSFER P&P1 Z-AXIS SAFETY PIN LOADING SENSOR", signal07 := "BK21"."X17-1 STACK NG BOX DETECT SENSOR", signal08 := "BK21"."X10-2 INS TRANSFER P&P1 Y-AXIS HOMING SENSOR", signal09 := "BK21"."X11-2 SPARE", signal10 := "BK21"."X12-2 INS TRANSFER P&P1 Z-AXIS HOMING SENSOR", signal11 := "BK21"."X13-2 SPARE", signal12 := "BK21"."X14-2 INS TRANSFER P&P1 CLAMP CLOSE SENSOR", signal13 := "BK21"."X15-2 INS TRANSFER P&P1 CLAMP OPEN/CLOSE PRESSURE SENSOR", signal14 := "BK21"."X16-2 SPARE", signal15 := "BK21"."X17-2 SPARE", interfaceSignals := "InstInterfaceSignals".statInterfaceSignalsHmi[23].valueSymbolLeft)
   END_RUNG
   // the same network as SCL:
   #instSignals23Left(signal00 := "BK21"."X10-1 INS TRANSFER P&P1 Y-AXIS LIMIT SENSOR(-)",   // "LAF_InterfaceSignalsBool"
                      signal01 := "BK21"."X11-1 INS TRANSFER P&P1 Y-AXIS LIMIT SENSOR(+)",
                      signal02 := "BK21"."X12-1 INS TRANSFER P&P1 Z-AXIS LIMIT SENSOR(-)",
                      signal03 := "BK21"."X13-1 INS TRANSFER P&P1 Z-AXIS LIMIT SENSOR(+)",
                      signal04 := "BK21"."X14-1 INS TRANSFER P&P1 CLAMP OPEN SENSOR",
                      signal05 := "BK21"."X15-1 INS TRANSFER P&P1 CLAMP STACK DETECT SENSOR",
                      signal06 := "BK21"."X16-1 INS TRANSFER P&P1 Z-AXIS SAFETY PIN LOADING SENSOR",
                      signal07 := "BK21"."X17-1 STACK NG BOX DETECT SENSOR",
                      signal08 := "BK21"."X10-2 INS TRANSFER P&P1 Y-AXIS HOMING SENSOR",
                      signal09 := "BK21"."X11-2 SPARE",
                      signal10 := "BK21"."X12-2 INS TRANSFER P&P1 Z-AXIS HOMING SENSOR",
                      signal11 := "BK21"."X13-2 SPARE",
                      signal12 := "BK21"."X14-2 INS TRANSFER P&P1 CLAMP CLOSE SENSOR",
                      signal13 := "BK21"."X15-2 INS TRANSFER P&P1 CLAMP OPEN/CLOSE PRESSURE SENSOR",
                      signal14 := "BK21"."X16-2 SPARE",
                      signal15 := "BK21"."X17-2 SPARE",
                      interfaceSignals := "InstInterfaceSignals".statInterfaceSignalsHmi[23].valueSymbolLeft);
END_REGION

REGION Network 29: Interface Signals 24 BK22
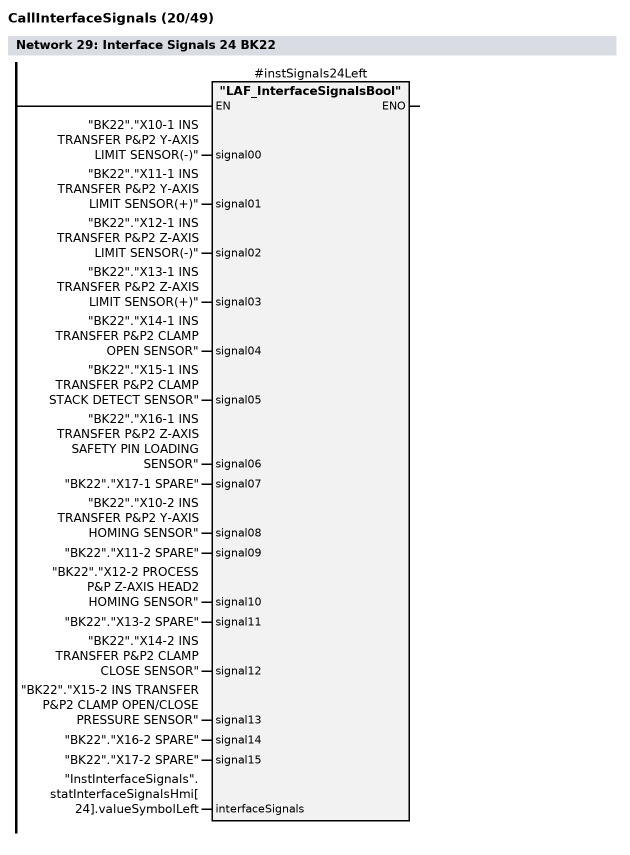
   RUNG wire#powerrail
      #instSignals24Left(signal00 := "BK22"."X10-1 INS TRANSFER P&P2 Y-AXIS LIMIT SENSOR(-)", signal01 := "BK22"."X11-1 INS TRANSFER P&P2 Y-AXIS LIMIT SENSOR(+)", signal02 := "BK22"."X12-1 INS TRANSFER P&P2 Z-AXIS LIMIT SENSOR(-)", signal03 := "BK22"."X13-1 INS TRANSFER P&P2 Z-AXIS LIMIT SENSOR(+)", signal04 := "BK22"."X14-1 INS TRANSFER P&P2 CLAMP OPEN SENSOR", signal05 := "BK22"."X15-1 INS TRANSFER P&P2 CLAMP STACK DETECT SENSOR", signal06 := "BK22"."X16-1 INS TRANSFER P&P2 Z-AXIS SAFETY PIN LOADING SENSOR", signal07 := "BK22"."X17-1 SPARE", signal08 := "BK22"."X10-2 INS TRANSFER P&P2 Y-AXIS HOMING SENSOR", signal09 := "BK22"."X11-2 SPARE", signal10 := "BK22"."X12-2 PROCESS P&P Z-AXIS HEAD2 HOMING SENSOR", signal11 := "BK22"."X13-2 SPARE", signal12 := "BK22"."X14-2 INS TRANSFER P&P2 CLAMP CLOSE SENSOR", signal13 := "BK22"."X15-2 INS TRANSFER P&P2 CLAMP OPEN/CLOSE PRESSURE SENSOR", signal14 := "BK22"."X16-2 SPARE", signal15 := "BK22"."X17-2 SPARE", interfaceSignals := "InstInterfaceSignals".statInterfaceSignalsHmi[24].valueSymbolLeft)
   END_RUNG
   // the same network as SCL:
   #instSignals24Left(signal00 := "BK22"."X10-1 INS TRANSFER P&P2 Y-AXIS LIMIT SENSOR(-)",   // "LAF_InterfaceSignalsBool"
                      signal01 := "BK22"."X11-1 INS TRANSFER P&P2 Y-AXIS LIMIT SENSOR(+)",
                      signal02 := "BK22"."X12-1 INS TRANSFER P&P2 Z-AXIS LIMIT SENSOR(-)",
                      signal03 := "BK22"."X13-1 INS TRANSFER P&P2 Z-AXIS LIMIT SENSOR(+)",
                      signal04 := "BK22"."X14-1 INS TRANSFER P&P2 CLAMP OPEN SENSOR",
                      signal05 := "BK22"."X15-1 INS TRANSFER P&P2 CLAMP STACK DETECT SENSOR",
                      signal06 := "BK22"."X16-1 INS TRANSFER P&P2 Z-AXIS SAFETY PIN LOADING SENSOR",
                      signal07 := "BK22"."X17-1 SPARE",
                      signal08 := "BK22"."X10-2 INS TRANSFER P&P2 Y-AXIS HOMING SENSOR",
                      signal09 := "BK22"."X11-2 SPARE",
                      signal10 := "BK22"."X12-2 PROCESS P&P Z-AXIS HEAD2 HOMING SENSOR",
                      signal11 := "BK22"."X13-2 SPARE",
                      signal12 := "BK22"."X14-2 INS TRANSFER P&P2 CLAMP CLOSE SENSOR",
                      signal13 := "BK22"."X15-2 INS TRANSFER P&P2 CLAMP OPEN/CLOSE PRESSURE SENSOR",
                      signal14 := "BK22"."X16-2 SPARE",
                      signal15 := "BK22"."X17-2 SPARE",
                      interfaceSignals := "InstInterfaceSignals".statInterfaceSignalsHmi[24].valueSymbolLeft);
END_REGION

REGION Network 30: Interface Signals 25 BK23
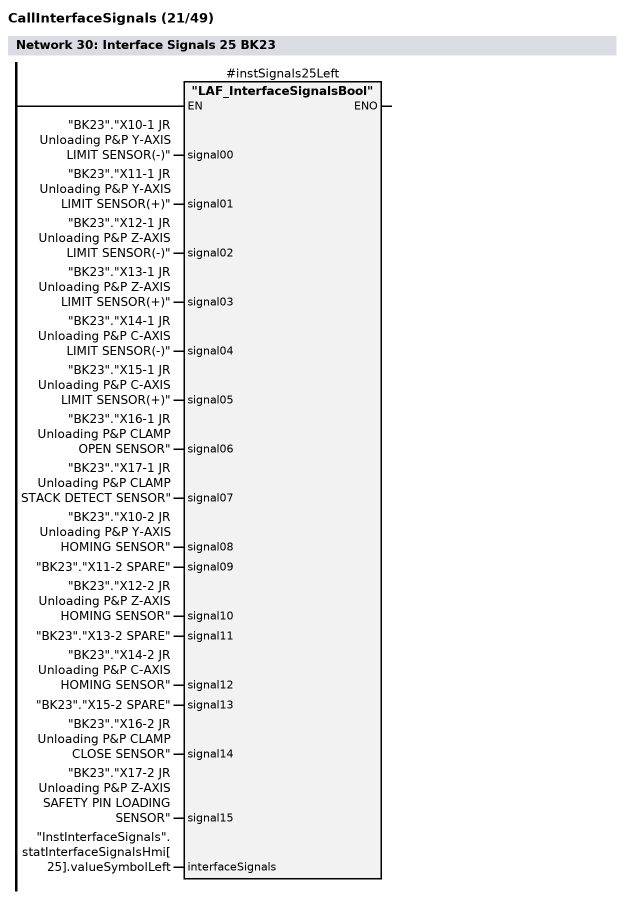
   RUNG wire#powerrail
      #instSignals25Left(signal00 := "BK23"."X10-1 JR Unloading P&P Y-AXIS LIMIT SENSOR(-)", signal01 := "BK23"."X11-1 JR Unloading P&P Y-AXIS LIMIT SENSOR(+)", signal02 := "BK23"."X12-1 JR Unloading P&P Z-AXIS LIMIT SENSOR(-)", signal03 := "BK23"."X13-1 JR Unloading P&P Z-AXIS LIMIT SENSOR(+)", signal04 := "BK23"."X14-1 JR Unloading P&P C-AXIS LIMIT SENSOR(-)", signal05 := "BK23"."X15-1 JR Unloading P&P C-AXIS LIMIT SENSOR(+)", signal06 := "BK23"."X16-1 JR Unloading P&P CLAMP OPEN SENSOR", signal07 := "BK23"."X17-1 JR Unloading P&P CLAMP STACK DETECT SENSOR", signal08 := "BK23"."X10-2 JR Unloading P&P Y-AXIS HOMING SENSOR", signal09 := "BK23"."X11-2 SPARE", signal10 := "BK23"."X12-2 JR Unloading P&P Z-AXIS HOMING SENSOR", signal11 := "BK23"."X13-2 SPARE", signal12 := "BK23"."X14-2 JR Unloading P&P C-AXIS HOMING SENSOR", signal13 := "BK23"."X15-2 SPARE", signal14 := "BK23"."X16-2 JR Unloading P&P CLAMP CLOSE SENSOR", signal15 := "BK23"."X17-2 JR Unloading P&P Z-AXIS SAFETY PIN LOADING SENSOR", interfaceSignals := "InstInterfaceSignals".statInterfaceSignalsHmi[25].valueSymbolLeft)
   END_RUNG
   // the same network as SCL:
   #instSignals25Left(signal00 := "BK23"."X10-1 JR Unloading P&P Y-AXIS LIMIT SENSOR(-)",   // "LAF_InterfaceSignalsBool"
                      signal01 := "BK23"."X11-1 JR Unloading P&P Y-AXIS LIMIT SENSOR(+)",
                      signal02 := "BK23"."X12-1 JR Unloading P&P Z-AXIS LIMIT SENSOR(-)",
                      signal03 := "BK23"."X13-1 JR Unloading P&P Z-AXIS LIMIT SENSOR(+)",
                      signal04 := "BK23"."X14-1 JR Unloading P&P C-AXIS LIMIT SENSOR(-)",
                      signal05 := "BK23"."X15-1 JR Unloading P&P C-AXIS LIMIT SENSOR(+)",
                      signal06 := "BK23"."X16-1 JR Unloading P&P CLAMP OPEN SENSOR",
                      signal07 := "BK23"."X17-1 JR Unloading P&P CLAMP STACK DETECT SENSOR",
                      signal08 := "BK23"."X10-2 JR Unloading P&P Y-AXIS HOMING SENSOR",
                      signal09 := "BK23"."X11-2 SPARE",
                      signal10 := "BK23"."X12-2 JR Unloading P&P Z-AXIS HOMING SENSOR",
                      signal11 := "BK23"."X13-2 SPARE",
                      signal12 := "BK23"."X14-2 JR Unloading P&P C-AXIS HOMING SENSOR",
                      signal13 := "BK23"."X15-2 SPARE",
                      signal14 := "BK23"."X16-2 JR Unloading P&P CLAMP CLOSE SENSOR",
                      signal15 := "BK23"."X17-2 JR Unloading P&P Z-AXIS SAFETY PIN LOADING SENSOR",
                      interfaceSignals := "InstInterfaceSignals".statInterfaceSignalsHmi[25].valueSymbolLeft);
END_REGION

REGION Network 31: Interface Signals 26 BK24
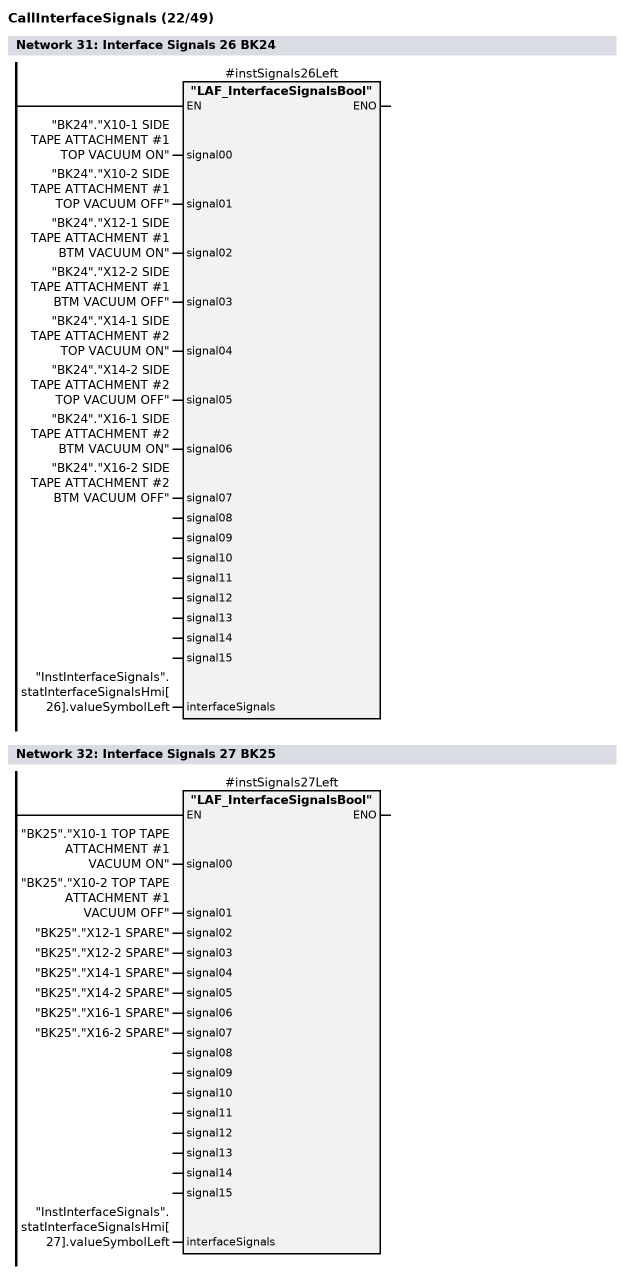
   RUNG wire#powerrail
      #instSignals26Left(signal00 := "BK24"."X10-1 SIDE TAPE ATTACHMENT #1 TOP VACUUM ON", signal01 := "BK24"."X10-2 SIDE TAPE ATTACHMENT #1 TOP VACUUM OFF", signal02 := "BK24"."X12-1 SIDE TAPE ATTACHMENT #1 BTM VACUUM ON", signal03 := "BK24"."X12-2 SIDE TAPE ATTACHMENT #1 BTM VACUUM OFF", signal04 := "BK24"."X14-1 SIDE TAPE ATTACHMENT #2 TOP VACUUM ON", signal05 := "BK24"."X14-2 SIDE TAPE ATTACHMENT #2 TOP VACUUM OFF", signal06 := "BK24"."X16-1 SIDE TAPE ATTACHMENT #2 BTM VACUUM ON", signal07 := "BK24"."X16-2 SIDE TAPE ATTACHMENT #2 BTM VACUUM OFF", signal08 :=, signal09 :=, signal10 :=, signal11 :=, signal12 :=, signal13 :=, signal14 :=, signal15 :=, interfaceSignals := "InstInterfaceSignals".statInterfaceSignalsHmi[26].valueSymbolLeft)
   END_RUNG
   // the same network as SCL:
   #instSignals26Left(signal00 := "BK24"."X10-1 SIDE TAPE ATTACHMENT #1 TOP VACUUM ON",   // "LAF_InterfaceSignalsBool"
                      signal01 := "BK24"."X10-2 SIDE TAPE ATTACHMENT #1 TOP VACUUM OFF",
                      signal02 := "BK24"."X12-1 SIDE TAPE ATTACHMENT #1 BTM VACUUM ON",
                      signal03 := "BK24"."X12-2 SIDE TAPE ATTACHMENT #1 BTM VACUUM OFF",
                      signal04 := "BK24"."X14-1 SIDE TAPE ATTACHMENT #2 TOP VACUUM ON",
                      signal05 := "BK24"."X14-2 SIDE TAPE ATTACHMENT #2 TOP VACUUM OFF",
                      signal06 := "BK24"."X16-1 SIDE TAPE ATTACHMENT #2 BTM VACUUM ON",
                      signal07 := "BK24"."X16-2 SIDE TAPE ATTACHMENT #2 BTM VACUUM OFF",
                      interfaceSignals := "InstInterfaceSignals".statInterfaceSignalsHmi[26].valueSymbolLeft);
END_REGION

REGION Network 32: Interface Signals 27 BK25
   RUNG wire#powerrail
      #instSignals27Left(signal00 := "BK25"."X10-1 TOP TAPE ATTACHMENT #1 VACUUM ON", signal01 := "BK25"."X10-2 TOP TAPE ATTACHMENT #1 VACUUM OFF", signal02 := "BK25"."X12-1 SPARE", signal03 := "BK25"."X12-2 SPARE", signal04 := "BK25"."X14-1 SPARE", signal05 := "BK25"."X14-2 SPARE", signal06 := "BK25"."X16-1 SPARE", signal07 := "BK25"."X16-2 SPARE", signal08 :=, signal09 :=, signal10 :=, signal11 :=, signal12 :=, signal13 :=, signal14 :=, signal15 :=, interfaceSignals := "InstInterfaceSignals".statInterfaceSignalsHmi[27].valueSymbolLeft)
   END_RUNG
   // the same network as SCL:
   #instSignals27Left(signal00 := "BK25"."X10-1 TOP TAPE ATTACHMENT #1 VACUUM ON",   // "LAF_InterfaceSignalsBool"
                      signal01 := "BK25"."X10-2 TOP TAPE ATTACHMENT #1 VACUUM OFF",
                      signal02 := "BK25"."X12-1 SPARE",
                      signal03 := "BK25"."X12-2 SPARE",
                      signal04 := "BK25"."X14-1 SPARE",
                      signal05 := "BK25"."X14-2 SPARE",
                      signal06 := "BK25"."X16-1 SPARE",
                      signal07 := "BK25"."X16-2 SPARE",
                      interfaceSignals := "InstInterfaceSignals".statInterfaceSignalsHmi[27].valueSymbolLeft);
END_REGION

REGION Network 33: Interface Signals 28 PM01
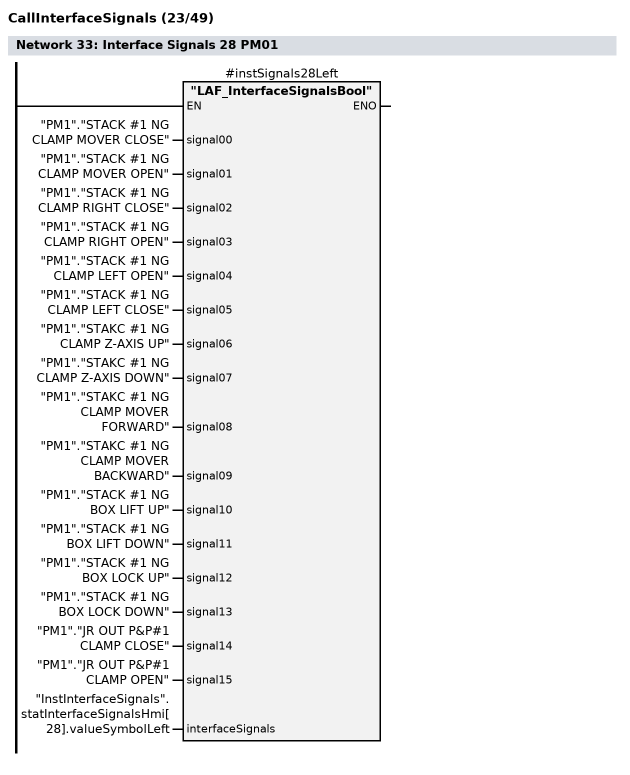
   RUNG wire#powerrail
      #instSignals28Left(signal00 := "PM1"."STACK #1 NG CLAMP MOVER CLOSE", signal01 := "PM1"."STACK #1 NG CLAMP MOVER OPEN", signal02 := "PM1"."STACK #1 NG CLAMP RIGHT CLOSE", signal03 := "PM1"."STACK #1 NG CLAMP RIGHT OPEN", signal04 := "PM1"."STACK #1 NG CLAMP LEFT OPEN", signal05 := "PM1"."STACK #1 NG CLAMP LEFT CLOSE", signal06 := "PM1"."STAKC #1 NG CLAMP Z-AXIS UP", signal07 := "PM1"."STAKC #1 NG CLAMP Z-AXIS DOWN", signal08 := "PM1"."STAKC #1 NG CLAMP MOVER FORWARD", signal09 := "PM1"."STAKC #1 NG CLAMP MOVER BACKWARD", signal10 := "PM1"."STACK #1 NG BOX LIFT UP", signal11 := "PM1"."STACK #1 NG BOX LIFT DOWN", signal12 := "PM1"."STACK #1 NG BOX LOCK UP", signal13 := "PM1"."STACK #1 NG BOX LOCK DOWN", signal14 := "PM1"."JR OUT P&P#1 CLAMP CLOSE", signal15 := "PM1"."JR OUT P&P#1 CLAMP OPEN", interfaceSignals := "InstInterfaceSignals".statInterfaceSignalsHmi[28].valueSymbolLeft)
   END_RUNG
   // the same network as SCL:
   #instSignals28Left(signal00 := "PM1"."STACK #1 NG CLAMP MOVER CLOSE",   // "LAF_InterfaceSignalsBool"
                      signal01 := "PM1"."STACK #1 NG CLAMP MOVER OPEN",
                      signal02 := "PM1"."STACK #1 NG CLAMP RIGHT CLOSE",
                      signal03 := "PM1"."STACK #1 NG CLAMP RIGHT OPEN",
                      signal04 := "PM1"."STACK #1 NG CLAMP LEFT OPEN",
                      signal05 := "PM1"."STACK #1 NG CLAMP LEFT CLOSE",
                      signal06 := "PM1"."STAKC #1 NG CLAMP Z-AXIS UP",
                      signal07 := "PM1"."STAKC #1 NG CLAMP Z-AXIS DOWN",
                      signal08 := "PM1"."STAKC #1 NG CLAMP MOVER FORWARD",
                      signal09 := "PM1"."STAKC #1 NG CLAMP MOVER BACKWARD",
                      signal10 := "PM1"."STACK #1 NG BOX LIFT UP",
                      signal11 := "PM1"."STACK #1 NG BOX LIFT DOWN",
                      signal12 := "PM1"."STACK #1 NG BOX LOCK UP",
                      signal13 := "PM1"."STACK #1 NG BOX LOCK DOWN",
                      signal14 := "PM1"."JR OUT P&P#1 CLAMP CLOSE",
                      signal15 := "PM1"."JR OUT P&P#1 CLAMP OPEN",
                      interfaceSignals := "InstInterfaceSignals".statInterfaceSignalsHmi[28].valueSymbolLeft);
END_REGION

REGION Network 34: Interface Signals 29 PM02
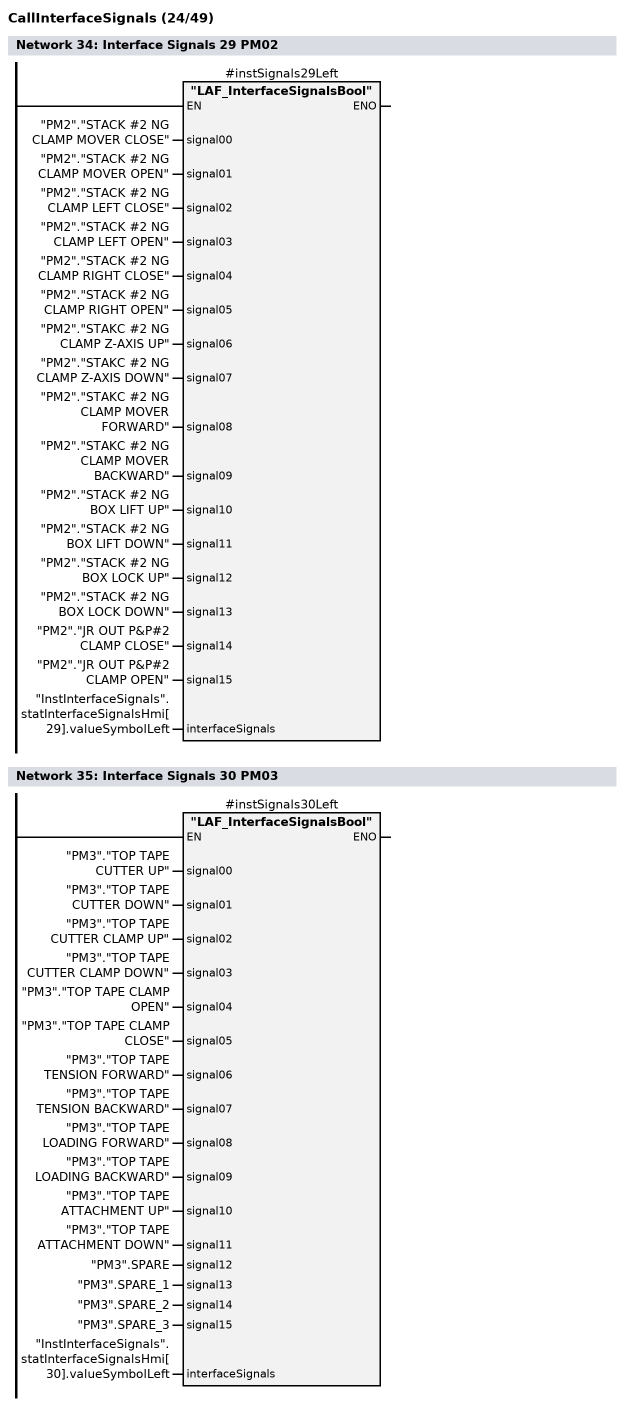
   RUNG wire#powerrail
      #instSignals29Left(signal00 := "PM2"."STACK #2 NG CLAMP MOVER CLOSE", signal01 := "PM2"."STACK #2 NG CLAMP MOVER OPEN", signal02 := "PM2"."STACK #2 NG CLAMP LEFT CLOSE", signal03 := "PM2"."STACK #2 NG CLAMP LEFT OPEN", signal04 := "PM2"."STACK #2 NG CLAMP RIGHT CLOSE", signal05 := "PM2"."STACK #2 NG CLAMP RIGHT OPEN", signal06 := "PM2"."STAKC #2 NG CLAMP Z-AXIS UP", signal07 := "PM2"."STAKC #2 NG CLAMP Z-AXIS DOWN", signal08 := "PM2"."STAKC #2 NG CLAMP MOVER FORWARD", signal09 := "PM2"."STAKC #2 NG CLAMP MOVER BACKWARD", signal10 := "PM2"."STACK #2 NG BOX LIFT UP", signal11 := "PM2"."STACK #2 NG BOX LIFT DOWN", signal12 := "PM2"."STACK #2 NG BOX LOCK UP", signal13 := "PM2"."STACK #2 NG BOX LOCK DOWN", signal14 := "PM2"."JR OUT P&P#2 CLAMP CLOSE", signal15 := "PM2"."JR OUT P&P#2 CLAMP OPEN", interfaceSignals := "InstInterfaceSignals".statInterfaceSignalsHmi[29].valueSymbolLeft)
   END_RUNG
   // the same network as SCL:
   #instSignals29Left(signal00 := "PM2"."STACK #2 NG CLAMP MOVER CLOSE",   // "LAF_InterfaceSignalsBool"
                      signal01 := "PM2"."STACK #2 NG CLAMP MOVER OPEN",
                      signal02 := "PM2"."STACK #2 NG CLAMP LEFT CLOSE",
                      signal03 := "PM2"."STACK #2 NG CLAMP LEFT OPEN",
                      signal04 := "PM2"."STACK #2 NG CLAMP RIGHT CLOSE",
                      signal05 := "PM2"."STACK #2 NG CLAMP RIGHT OPEN",
                      signal06 := "PM2"."STAKC #2 NG CLAMP Z-AXIS UP",
                      signal07 := "PM2"."STAKC #2 NG CLAMP Z-AXIS DOWN",
                      signal08 := "PM2"."STAKC #2 NG CLAMP MOVER FORWARD",
                      signal09 := "PM2"."STAKC #2 NG CLAMP MOVER BACKWARD",
                      signal10 := "PM2"."STACK #2 NG BOX LIFT UP",
                      signal11 := "PM2"."STACK #2 NG BOX LIFT DOWN",
                      signal12 := "PM2"."STACK #2 NG BOX LOCK UP",
                      signal13 := "PM2"."STACK #2 NG BOX LOCK DOWN",
                      signal14 := "PM2"."JR OUT P&P#2 CLAMP CLOSE",
                      signal15 := "PM2"."JR OUT P&P#2 CLAMP OPEN",
                      interfaceSignals := "InstInterfaceSignals".statInterfaceSignalsHmi[29].valueSymbolLeft);
END_REGION

REGION Network 35: Interface Signals 30 PM03
   RUNG wire#powerrail
      #instSignals30Left(signal00 := "PM3"."TOP TAPE CUTTER UP", signal01 := "PM3"."TOP TAPE CUTTER DOWN", signal02 := "PM3"."TOP TAPE CUTTER CLAMP UP", signal03 := "PM3"."TOP TAPE CUTTER CLAMP DOWN", signal04 := "PM3"."TOP TAPE CLAMP OPEN", signal05 := "PM3"."TOP TAPE CLAMP CLOSE", signal06 := "PM3"."TOP TAPE TENSION FORWARD", signal07 := "PM3"."TOP TAPE TENSION BACKWARD", signal08 := "PM3"."TOP TAPE LOADING FORWARD", signal09 := "PM3"."TOP TAPE LOADING BACKWARD", signal10 := "PM3"."TOP TAPE ATTACHMENT UP", signal11 := "PM3"."TOP TAPE ATTACHMENT DOWN", signal12 := "PM3".SPARE, signal13 := "PM3".SPARE_1, signal14 := "PM3".SPARE_2, signal15 := "PM3".SPARE_3, interfaceSignals := "InstInterfaceSignals".statInterfaceSignalsHmi[30].valueSymbolLeft)
   END_RUNG
   // the same network as SCL:
   #instSignals30Left(signal00 := "PM3"."TOP TAPE CUTTER UP",   // "LAF_InterfaceSignalsBool"
                      signal01 := "PM3"."TOP TAPE CUTTER DOWN",
                      signal02 := "PM3"."TOP TAPE CUTTER CLAMP UP",
                      signal03 := "PM3"."TOP TAPE CUTTER CLAMP DOWN",
                      signal04 := "PM3"."TOP TAPE CLAMP OPEN",
                      signal05 := "PM3"."TOP TAPE CLAMP CLOSE",
                      signal06 := "PM3"."TOP TAPE TENSION FORWARD",
                      signal07 := "PM3"."TOP TAPE TENSION BACKWARD",
                      signal08 := "PM3"."TOP TAPE LOADING FORWARD",
                      signal09 := "PM3"."TOP TAPE LOADING BACKWARD",
                      signal10 := "PM3"."TOP TAPE ATTACHMENT UP",
                      signal11 := "PM3"."TOP TAPE ATTACHMENT DOWN",
                      signal12 := "PM3".SPARE,
                      signal13 := "PM3".SPARE_1,
                      signal14 := "PM3".SPARE_2,
                      signal15 := "PM3".SPARE_3,
                      interfaceSignals := "InstInterfaceSignals".statInterfaceSignalsHmi[30].valueSymbolLeft);
END_REGION

REGION Network 36: Interface Signals 31 PM04
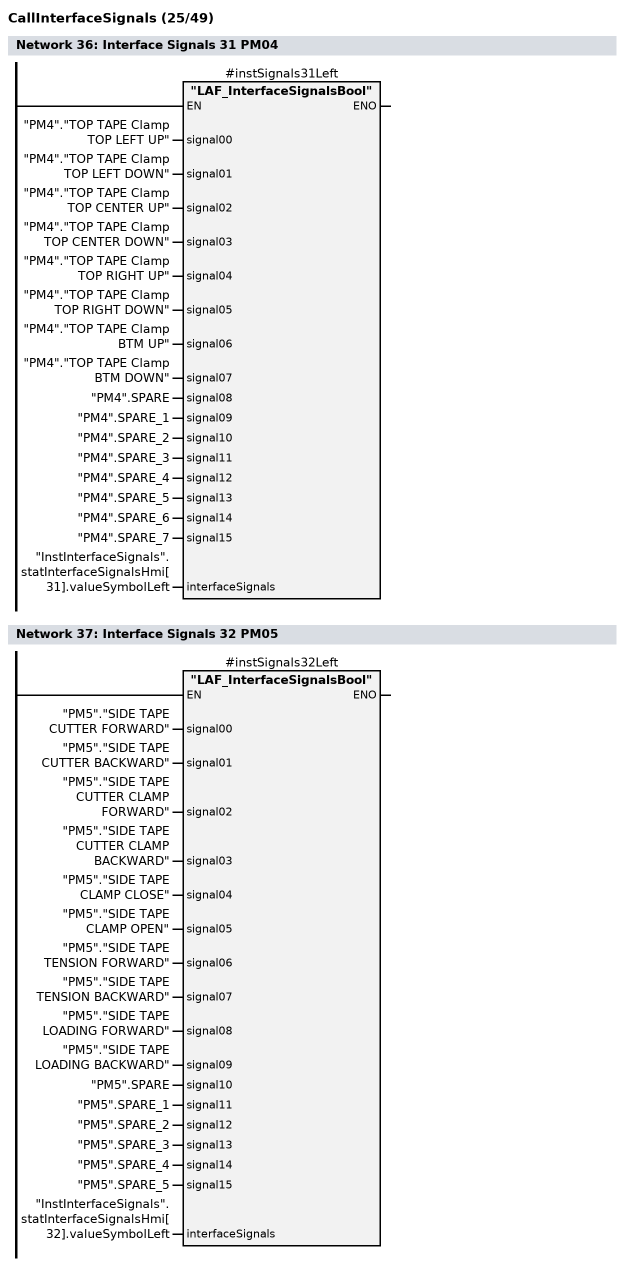
   RUNG wire#powerrail
      #instSignals31Left(signal00 := "PM4"."TOP TAPE Clamp TOP LEFT UP", signal01 := "PM4"."TOP TAPE Clamp TOP LEFT DOWN", signal02 := "PM4"."TOP TAPE Clamp TOP CENTER UP", signal03 := "PM4"."TOP TAPE Clamp TOP CENTER DOWN", signal04 := "PM4"."TOP TAPE Clamp TOP RIGHT UP", signal05 := "PM4"."TOP TAPE Clamp TOP RIGHT DOWN", signal06 := "PM4"."TOP TAPE Clamp BTM UP", signal07 := "PM4"."TOP TAPE Clamp BTM DOWN", signal08 := "PM4".SPARE, signal09 := "PM4".SPARE_1, signal10 := "PM4".SPARE_2, signal11 := "PM4".SPARE_3, signal12 := "PM4".SPARE_4, signal13 := "PM4".SPARE_5, signal14 := "PM4".SPARE_6, signal15 := "PM4".SPARE_7, interfaceSignals := "InstInterfaceSignals".statInterfaceSignalsHmi[31].valueSymbolLeft)
   END_RUNG
   // the same network as SCL:
   #instSignals31Left(signal00 := "PM4"."TOP TAPE Clamp TOP LEFT UP",   // "LAF_InterfaceSignalsBool"
                      signal01 := "PM4"."TOP TAPE Clamp TOP LEFT DOWN",
                      signal02 := "PM4"."TOP TAPE Clamp TOP CENTER UP",
                      signal03 := "PM4"."TOP TAPE Clamp TOP CENTER DOWN",
                      signal04 := "PM4"."TOP TAPE Clamp TOP RIGHT UP",
                      signal05 := "PM4"."TOP TAPE Clamp TOP RIGHT DOWN",
                      signal06 := "PM4"."TOP TAPE Clamp BTM UP",
                      signal07 := "PM4"."TOP TAPE Clamp BTM DOWN",
                      signal08 := "PM4".SPARE,
                      signal09 := "PM4".SPARE_1,
                      signal10 := "PM4".SPARE_2,
                      signal11 := "PM4".SPARE_3,
                      signal12 := "PM4".SPARE_4,
                      signal13 := "PM4".SPARE_5,
                      signal14 := "PM4".SPARE_6,
                      signal15 := "PM4".SPARE_7,
                      interfaceSignals := "InstInterfaceSignals".statInterfaceSignalsHmi[31].valueSymbolLeft);
END_REGION

REGION Network 37: Interface Signals 32 PM05
   RUNG wire#powerrail
      #instSignals32Left(signal00 := "PM5"."SIDE TAPE CUTTER FORWARD", signal01 := "PM5"."SIDE TAPE CUTTER BACKWARD", signal02 := "PM5"."SIDE TAPE CUTTER CLAMP FORWARD", signal03 := "PM5"."SIDE TAPE CUTTER CLAMP BACKWARD", signal04 := "PM5"."SIDE TAPE CLAMP CLOSE", signal05 := "PM5"."SIDE TAPE CLAMP OPEN", signal06 := "PM5"."SIDE TAPE TENSION FORWARD", signal07 := "PM5"."SIDE TAPE TENSION BACKWARD", signal08 := "PM5"."SIDE TAPE LOADING FORWARD", signal09 := "PM5"."SIDE TAPE LOADING BACKWARD", signal10 := "PM5".SPARE, signal11 := "PM5".SPARE_1, signal12 := "PM5".SPARE_2, signal13 := "PM5".SPARE_3, signal14 := "PM5".SPARE_4, signal15 := "PM5".SPARE_5, interfaceSignals := "InstInterfaceSignals".statInterfaceSignalsHmi[32].valueSymbolLeft)
   END_RUNG
   // the same network as SCL:
   #instSignals32Left(signal00 := "PM5"."SIDE TAPE CUTTER FORWARD",   // "LAF_InterfaceSignalsBool"
                      signal01 := "PM5"."SIDE TAPE CUTTER BACKWARD",
                      signal02 := "PM5"."SIDE TAPE CUTTER CLAMP FORWARD",
                      signal03 := "PM5"."SIDE TAPE CUTTER CLAMP BACKWARD",
                      signal04 := "PM5"."SIDE TAPE CLAMP CLOSE",
                      signal05 := "PM5"."SIDE TAPE CLAMP OPEN",
                      signal06 := "PM5"."SIDE TAPE TENSION FORWARD",
                      signal07 := "PM5"."SIDE TAPE TENSION BACKWARD",
                      signal08 := "PM5"."SIDE TAPE LOADING FORWARD",
                      signal09 := "PM5"."SIDE TAPE LOADING BACKWARD",
                      signal10 := "PM5".SPARE,
                      signal11 := "PM5".SPARE_1,
                      signal12 := "PM5".SPARE_2,
                      signal13 := "PM5".SPARE_3,
                      signal14 := "PM5".SPARE_4,
                      signal15 := "PM5".SPARE_5,
                      interfaceSignals := "InstInterfaceSignals".statInterfaceSignalsHmi[32].valueSymbolLeft);
END_REGION

REGION Network 38: Interface Signals 33 PM06
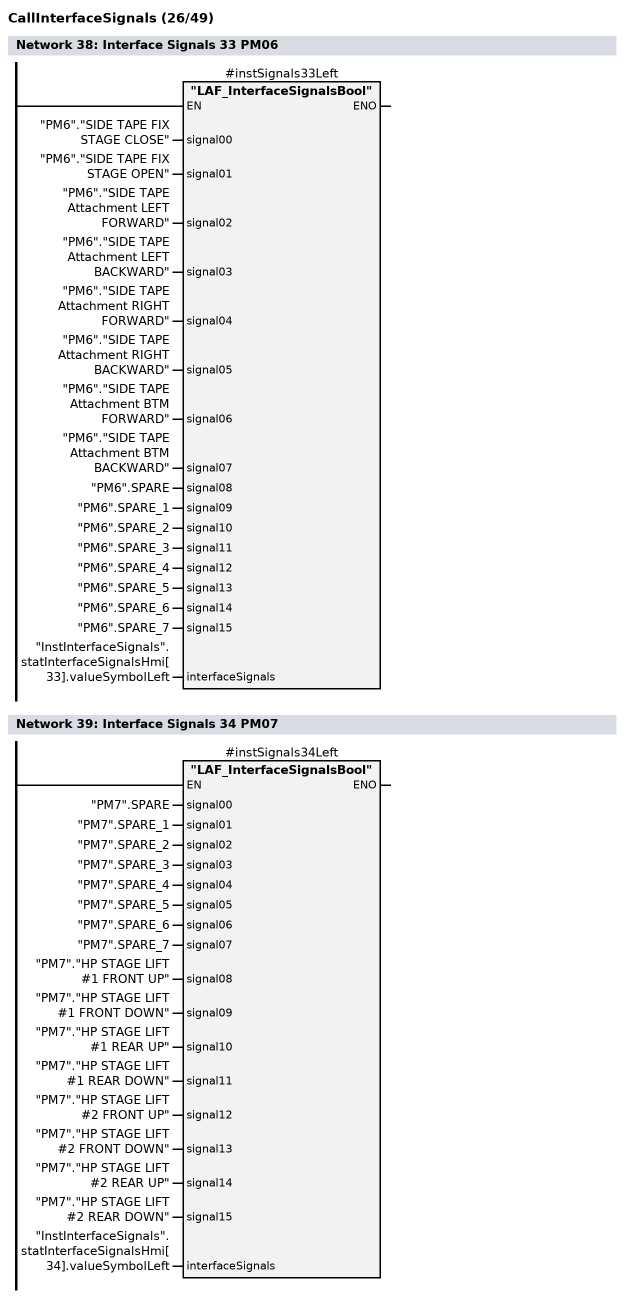
   RUNG wire#powerrail
      #instSignals33Left(signal00 := "PM6"."SIDE TAPE FIX STAGE CLOSE", signal01 := "PM6"."SIDE TAPE FIX STAGE OPEN", signal02 := "PM6"."SIDE TAPE Attachment LEFT FORWARD", signal03 := "PM6"."SIDE TAPE Attachment LEFT BACKWARD", signal04 := "PM6"."SIDE TAPE Attachment RIGHT FORWARD", signal05 := "PM6"."SIDE TAPE Attachment RIGHT BACKWARD", signal06 := "PM6"."SIDE TAPE Attachment BTM FORWARD", signal07 := "PM6"."SIDE TAPE Attachment BTM BACKWARD", signal08 := "PM6".SPARE, signal09 := "PM6".SPARE_1, signal10 := "PM6".SPARE_2, signal11 := "PM6".SPARE_3, signal12 := "PM6".SPARE_4, signal13 := "PM6".SPARE_5, signal14 := "PM6".SPARE_6, signal15 := "PM6".SPARE_7, interfaceSignals := "InstInterfaceSignals".statInterfaceSignalsHmi[33].valueSymbolLeft)
   END_RUNG
   // the same network as SCL:
   #instSignals33Left(signal00 := "PM6"."SIDE TAPE FIX STAGE CLOSE",   // "LAF_InterfaceSignalsBool"
                      signal01 := "PM6"."SIDE TAPE FIX STAGE OPEN",
                      signal02 := "PM6"."SIDE TAPE Attachment LEFT FORWARD",
                      signal03 := "PM6"."SIDE TAPE Attachment LEFT BACKWARD",
                      signal04 := "PM6"."SIDE TAPE Attachment RIGHT FORWARD",
                      signal05 := "PM6"."SIDE TAPE Attachment RIGHT BACKWARD",
                      signal06 := "PM6"."SIDE TAPE Attachment BTM FORWARD",
                      signal07 := "PM6"."SIDE TAPE Attachment BTM BACKWARD",
                      signal08 := "PM6".SPARE,
                      signal09 := "PM6".SPARE_1,
                      signal10 := "PM6".SPARE_2,
                      signal11 := "PM6".SPARE_3,
                      signal12 := "PM6".SPARE_4,
                      signal13 := "PM6".SPARE_5,
                      signal14 := "PM6".SPARE_6,
                      signal15 := "PM6".SPARE_7,
                      interfaceSignals := "InstInterfaceSignals".statInterfaceSignalsHmi[33].valueSymbolLeft);
END_REGION

REGION Network 39: Interface Signals 34 PM07
   RUNG wire#powerrail
      #instSignals34Left(signal00 := "PM7".SPARE, signal01 := "PM7".SPARE_1, signal02 := "PM7".SPARE_2, signal03 := "PM7".SPARE_3, signal04 := "PM7".SPARE_4, signal05 := "PM7".SPARE_5, signal06 := "PM7".SPARE_6, signal07 := "PM7".SPARE_7, signal08 := "PM7"."HP STAGE LIFT #1 FRONT UP", signal09 := "PM7"."HP STAGE LIFT #1 FRONT DOWN", signal10 := "PM7"."HP STAGE LIFT #1 REAR UP", signal11 := "PM7"."HP STAGE LIFT #1 REAR DOWN", signal12 := "PM7"."HP STAGE LIFT #2 FRONT UP", signal13 := "PM7"."HP STAGE LIFT #2 FRONT DOWN", signal14 := "PM7"."HP STAGE LIFT #2 REAR UP", signal15 := "PM7"."HP STAGE LIFT #2 REAR DOWN", interfaceSignals := "InstInterfaceSignals".statInterfaceSignalsHmi[34].valueSymbolLeft)
   END_RUNG
   // the same network as SCL:
   #instSignals34Left(signal00 := "PM7".SPARE,   // "LAF_InterfaceSignalsBool"
                      signal01 := "PM7".SPARE_1,
                      signal02 := "PM7".SPARE_2,
                      signal03 := "PM7".SPARE_3,
                      signal04 := "PM7".SPARE_4,
                      signal05 := "PM7".SPARE_5,
                      signal06 := "PM7".SPARE_6,
                      signal07 := "PM7".SPARE_7,
                      signal08 := "PM7"."HP STAGE LIFT #1 FRONT UP",
                      signal09 := "PM7"."HP STAGE LIFT #1 FRONT DOWN",
                      signal10 := "PM7"."HP STAGE LIFT #1 REAR UP",
                      signal11 := "PM7"."HP STAGE LIFT #1 REAR DOWN",
                      signal12 := "PM7"."HP STAGE LIFT #2 FRONT UP",
                      signal13 := "PM7"."HP STAGE LIFT #2 FRONT DOWN",
                      signal14 := "PM7"."HP STAGE LIFT #2 REAR UP",
                      signal15 := "PM7"."HP STAGE LIFT #2 REAR DOWN",
                      interfaceSignals := "InstInterfaceSignals".statInterfaceSignalsHmi[34].valueSymbolLeft);
END_REGION

REGION Network 40: Interface Signals 35 PM08
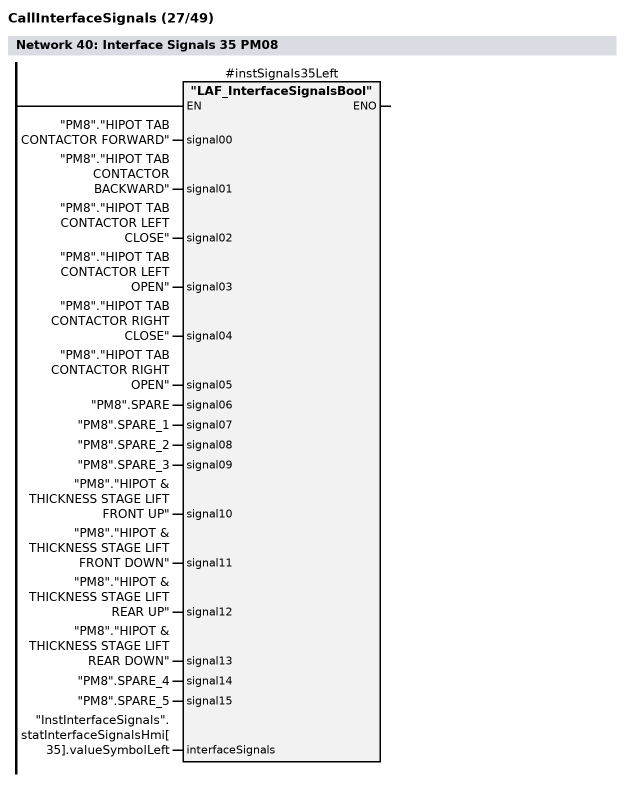
   RUNG wire#powerrail
      #instSignals35Left(signal00 := "PM8"."HIPOT TAB CONTACTOR FORWARD", signal01 := "PM8"."HIPOT TAB CONTACTOR BACKWARD", signal02 := "PM8"."HIPOT TAB CONTACTOR LEFT CLOSE", signal03 := "PM8"."HIPOT TAB CONTACTOR LEFT OPEN", signal04 := "PM8"."HIPOT TAB CONTACTOR RIGHT CLOSE", signal05 := "PM8"."HIPOT TAB CONTACTOR RIGHT OPEN", signal06 := "PM8".SPARE, signal07 := "PM8".SPARE_1, signal08 := "PM8".SPARE_2, signal09 := "PM8".SPARE_3, signal10 := "PM8"."HIPOT & THICKNESS STAGE LIFT FRONT UP", signal11 := "PM8"."HIPOT & THICKNESS STAGE LIFT FRONT DOWN", signal12 := "PM8"."HIPOT & THICKNESS STAGE LIFT REAR UP", signal13 := "PM8"."HIPOT & THICKNESS STAGE LIFT REAR DOWN", signal14 := "PM8".SPARE_4, signal15 := "PM8".SPARE_5, interfaceSignals := "InstInterfaceSignals".statInterfaceSignalsHmi[35].valueSymbolLeft)
   END_RUNG
   // the same network as SCL:
   #instSignals35Left(signal00 := "PM8"."HIPOT TAB CONTACTOR FORWARD",   // "LAF_InterfaceSignalsBool"
                      signal01 := "PM8"."HIPOT TAB CONTACTOR BACKWARD",
                      signal02 := "PM8"."HIPOT TAB CONTACTOR LEFT CLOSE",
                      signal03 := "PM8"."HIPOT TAB CONTACTOR LEFT OPEN",
                      signal04 := "PM8"."HIPOT TAB CONTACTOR RIGHT CLOSE",
                      signal05 := "PM8"."HIPOT TAB CONTACTOR RIGHT OPEN",
                      signal06 := "PM8".SPARE,
                      signal07 := "PM8".SPARE_1,
                      signal08 := "PM8".SPARE_2,
                      signal09 := "PM8".SPARE_3,
                      signal10 := "PM8"."HIPOT & THICKNESS STAGE LIFT FRONT UP",
                      signal11 := "PM8"."HIPOT & THICKNESS STAGE LIFT FRONT DOWN",
                      signal12 := "PM8"."HIPOT & THICKNESS STAGE LIFT REAR UP",
                      signal13 := "PM8"."HIPOT & THICKNESS STAGE LIFT REAR DOWN",
                      signal14 := "PM8".SPARE_4,
                      signal15 := "PM8".SPARE_5,
                      interfaceSignals := "InstInterfaceSignals".statInterfaceSignalsHmi[35].valueSymbolLeft);
END_REGION

REGION Network 41: Interface Signals 36 PM09
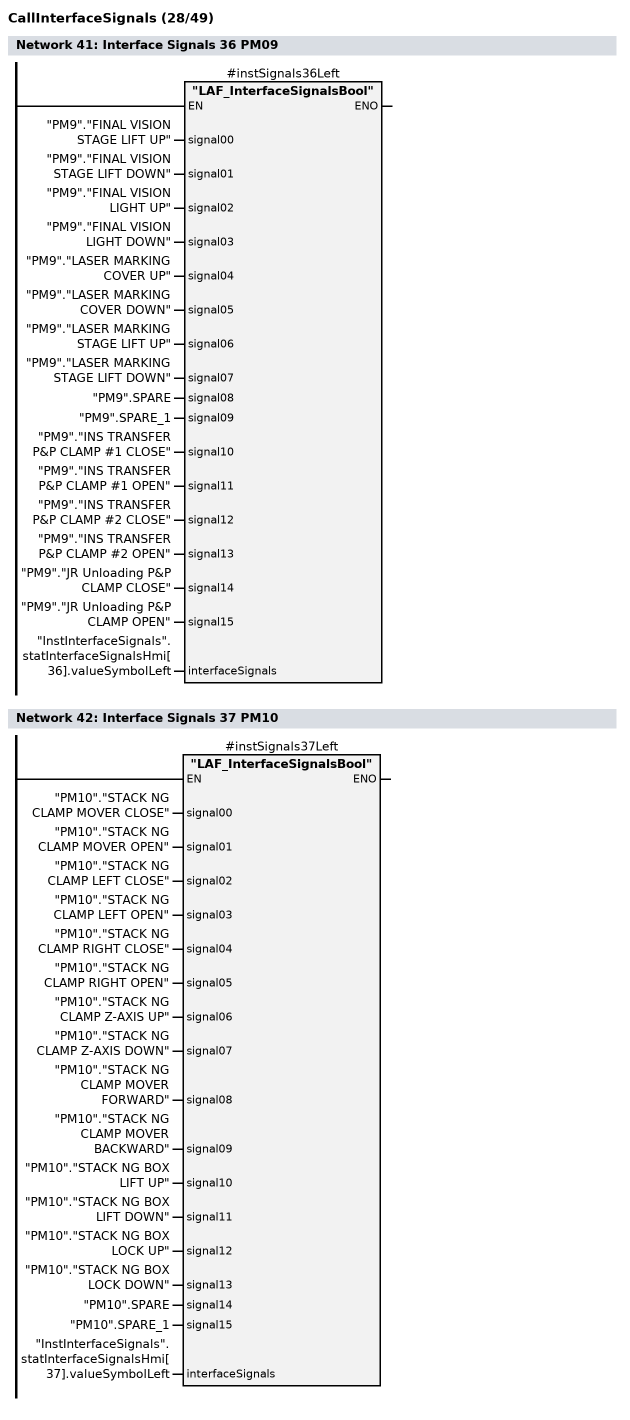
   RUNG wire#powerrail
      #instSignals36Left(signal00 := "PM9"."FINAL VISION STAGE LIFT UP", signal01 := "PM9"."FINAL VISION STAGE LIFT DOWN", signal02 := "PM9"."FINAL VISION LIGHT UP", signal03 := "PM9"."FINAL VISION LIGHT DOWN", signal04 := "PM9"."LASER MARKING COVER UP", signal05 := "PM9"."LASER MARKING COVER DOWN", signal06 := "PM9"."LASER MARKING STAGE LIFT UP", signal07 := "PM9"."LASER MARKING STAGE LIFT DOWN", signal08 := "PM9".SPARE, signal09 := "PM9".SPARE_1, signal10 := "PM9"."INS TRANSFER P&P CLAMP #1 CLOSE", signal11 := "PM9"."INS TRANSFER P&P CLAMP #1 OPEN", signal12 := "PM9"."INS TRANSFER P&P CLAMP #2 CLOSE", signal13 := "PM9"."INS TRANSFER P&P CLAMP #2 OPEN", signal14 := "PM9"."JR Unloading P&P CLAMP CLOSE", signal15 := "PM9"."JR Unloading P&P CLAMP OPEN", interfaceSignals := "InstInterfaceSignals".statInterfaceSignalsHmi[36].valueSymbolLeft)
   END_RUNG
   // the same network as SCL:
   #instSignals36Left(signal00 := "PM9"."FINAL VISION STAGE LIFT UP",   // "LAF_InterfaceSignalsBool"
                      signal01 := "PM9"."FINAL VISION STAGE LIFT DOWN",
                      signal02 := "PM9"."FINAL VISION LIGHT UP",
                      signal03 := "PM9"."FINAL VISION LIGHT DOWN",
                      signal04 := "PM9"."LASER MARKING COVER UP",
                      signal05 := "PM9"."LASER MARKING COVER DOWN",
                      signal06 := "PM9"."LASER MARKING STAGE LIFT UP",
                      signal07 := "PM9"."LASER MARKING STAGE LIFT DOWN",
                      signal08 := "PM9".SPARE,
                      signal09 := "PM9".SPARE_1,
                      signal10 := "PM9"."INS TRANSFER P&P CLAMP #1 CLOSE",
                      signal11 := "PM9"."INS TRANSFER P&P CLAMP #1 OPEN",
                      signal12 := "PM9"."INS TRANSFER P&P CLAMP #2 CLOSE",
                      signal13 := "PM9"."INS TRANSFER P&P CLAMP #2 OPEN",
                      signal14 := "PM9"."JR Unloading P&P CLAMP CLOSE",
                      signal15 := "PM9"."JR Unloading P&P CLAMP OPEN",
                      interfaceSignals := "InstInterfaceSignals".statInterfaceSignalsHmi[36].valueSymbolLeft);
END_REGION

REGION Network 42: Interface Signals 37 PM10
   RUNG wire#powerrail
      #instSignals37Left(signal00 := "PM10"."STACK NG CLAMP MOVER CLOSE", signal01 := "PM10"."STACK NG CLAMP MOVER OPEN", signal02 := "PM10"."STACK NG CLAMP LEFT CLOSE", signal03 := "PM10"."STACK NG CLAMP LEFT OPEN", signal04 := "PM10"."STACK NG CLAMP RIGHT CLOSE", signal05 := "PM10"."STACK NG CLAMP RIGHT OPEN", signal06 := "PM10"."STACK NG CLAMP Z-AXIS UP", signal07 := "PM10"."STACK NG CLAMP Z-AXIS DOWN", signal08 := "PM10"."STACK NG CLAMP MOVER FORWARD", signal09 := "PM10"."STACK NG CLAMP MOVER BACKWARD", signal10 := "PM10"."STACK NG BOX LIFT UP", signal11 := "PM10"."STACK NG BOX LIFT DOWN", signal12 := "PM10"."STACK NG BOX LOCK UP", signal13 := "PM10"."STACK NG BOX LOCK DOWN", signal14 := "PM10".SPARE, signal15 := "PM10".SPARE_1, interfaceSignals := "InstInterfaceSignals".statInterfaceSignalsHmi[37].valueSymbolLeft)
   END_RUNG
   // the same network as SCL:
   #instSignals37Left(signal00 := "PM10"."STACK NG CLAMP MOVER CLOSE",   // "LAF_InterfaceSignalsBool"
                      signal01 := "PM10"."STACK NG CLAMP MOVER OPEN",
                      signal02 := "PM10"."STACK NG CLAMP LEFT CLOSE",
                      signal03 := "PM10"."STACK NG CLAMP LEFT OPEN",
                      signal04 := "PM10"."STACK NG CLAMP RIGHT CLOSE",
                      signal05 := "PM10"."STACK NG CLAMP RIGHT OPEN",
                      signal06 := "PM10"."STACK NG CLAMP Z-AXIS UP",
                      signal07 := "PM10"."STACK NG CLAMP Z-AXIS DOWN",
                      signal08 := "PM10"."STACK NG CLAMP MOVER FORWARD",
                      signal09 := "PM10"."STACK NG CLAMP MOVER BACKWARD",
                      signal10 := "PM10"."STACK NG BOX LIFT UP",
                      signal11 := "PM10"."STACK NG BOX LIFT DOWN",
                      signal12 := "PM10"."STACK NG BOX LOCK UP",
                      signal13 := "PM10"."STACK NG BOX LOCK DOWN",
                      signal14 := "PM10".SPARE,
                      signal15 := "PM10".SPARE_1,
                      interfaceSignals := "InstInterfaceSignals".statInterfaceSignalsHmi[37].valueSymbolLeft);
END_REGION

REGION Network 43: Interface Signals 38 SBK01
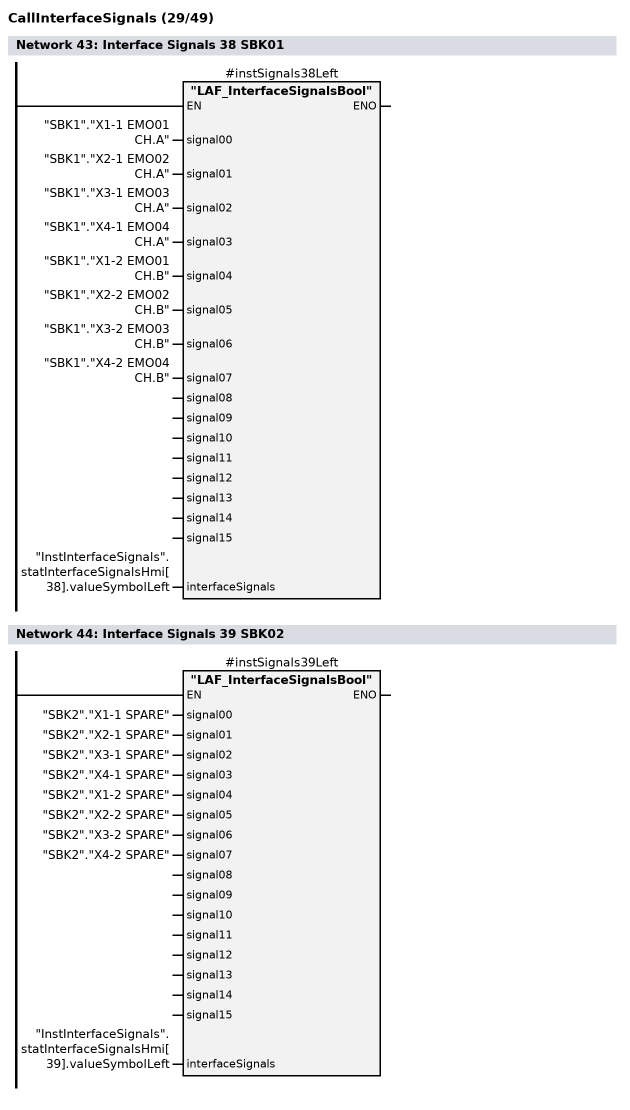
   RUNG wire#powerrail
      #instSignals38Left(signal00 := "SBK1"."X1-1 EMO01 CH.A", signal01 := "SBK1"."X2-1 EMO02 CH.A", signal02 := "SBK1"."X3-1 EMO03 CH.A", signal03 := "SBK1"."X4-1 EMO04 CH.A", signal04 := "SBK1"."X1-2 EMO01 CH.B", signal05 := "SBK1"."X2-2 EMO02 CH.B", signal06 := "SBK1"."X3-2 EMO03 CH.B", signal07 := "SBK1"."X4-2 EMO04 CH.B", signal08 :=, signal09 :=, signal10 :=, signal11 :=, signal12 :=, signal13 :=, signal14 :=, signal15 :=, interfaceSignals := "InstInterfaceSignals".statInterfaceSignalsHmi[38].valueSymbolLeft)
   END_RUNG
   // the same network as SCL:
   #instSignals38Left(signal00 := "SBK1"."X1-1 EMO01 CH.A",   // "LAF_InterfaceSignalsBool"
                      signal01 := "SBK1"."X2-1 EMO02 CH.A",
                      signal02 := "SBK1"."X3-1 EMO03 CH.A",
                      signal03 := "SBK1"."X4-1 EMO04 CH.A",
                      signal04 := "SBK1"."X1-2 EMO01 CH.B",
                      signal05 := "SBK1"."X2-2 EMO02 CH.B",
                      signal06 := "SBK1"."X3-2 EMO03 CH.B",
                      signal07 := "SBK1"."X4-2 EMO04 CH.B",
                      interfaceSignals := "InstInterfaceSignals".statInterfaceSignalsHmi[38].valueSymbolLeft);
END_REGION

REGION Network 44: Interface Signals 39 SBK02
   RUNG wire#powerrail
      #instSignals39Left(signal00 := "SBK2"."X1-1 SPARE", signal01 := "SBK2"."X2-1 SPARE", signal02 := "SBK2"."X3-1 SPARE", signal03 := "SBK2"."X4-1 SPARE", signal04 := "SBK2"."X1-2 SPARE", signal05 := "SBK2"."X2-2 SPARE", signal06 := "SBK2"."X3-2 SPARE", signal07 := "SBK2"."X4-2 SPARE", signal08 :=, signal09 :=, signal10 :=, signal11 :=, signal12 :=, signal13 :=, signal14 :=, signal15 :=, interfaceSignals := "InstInterfaceSignals".statInterfaceSignalsHmi[39].valueSymbolLeft)
   END_RUNG
   // the same network as SCL:
   #instSignals39Left(signal00 := "SBK2"."X1-1 SPARE",   // "LAF_InterfaceSignalsBool"
                      signal01 := "SBK2"."X2-1 SPARE",
                      signal02 := "SBK2"."X3-1 SPARE",
                      signal03 := "SBK2"."X4-1 SPARE",
                      signal04 := "SBK2"."X1-2 SPARE",
                      signal05 := "SBK2"."X2-2 SPARE",
                      signal06 := "SBK2"."X3-2 SPARE",
                      signal07 := "SBK2"."X4-2 SPARE",
                      interfaceSignals := "InstInterfaceSignals".statInterfaceSignalsHmi[39].valueSymbolLeft);
END_REGION

REGION Network 45: Interface Signals 40 SBK03
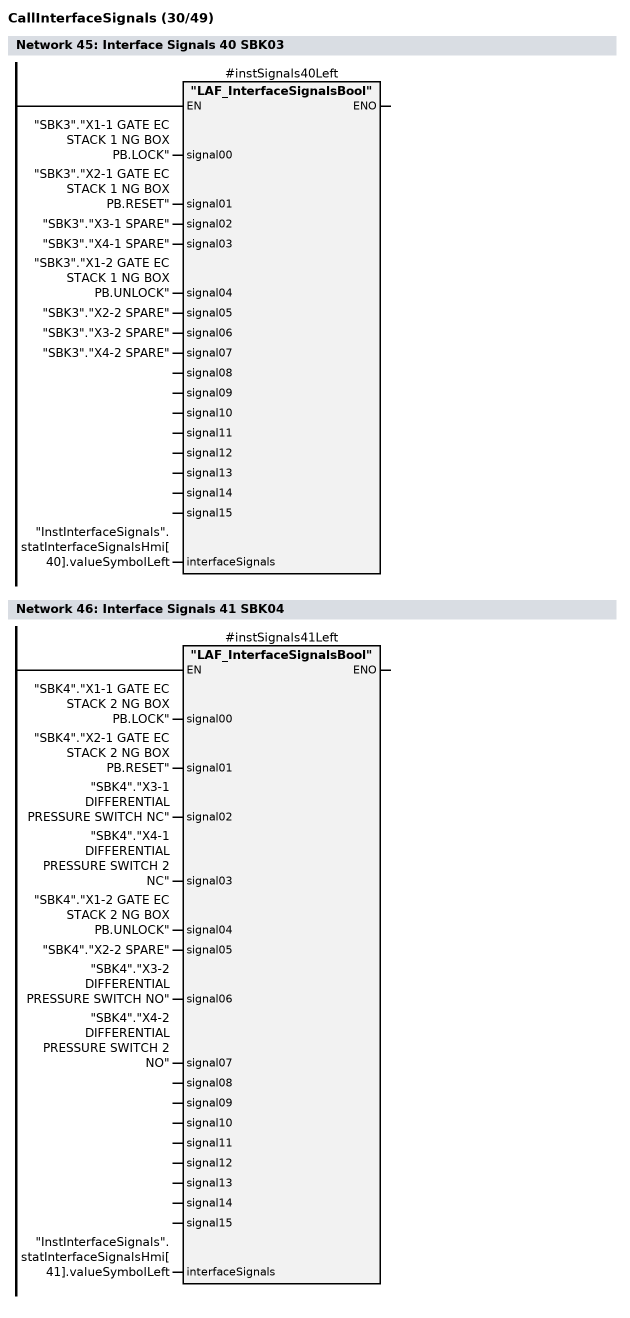
   RUNG wire#powerrail
      #instSignals40Left(signal00 := "SBK3"."X1-1 GATE EC STACK 1 NG BOX PB.LOCK", signal01 := "SBK3"."X2-1 GATE EC STACK 1 NG BOX PB.RESET", signal02 := "SBK3"."X3-1 SPARE", signal03 := "SBK3"."X4-1 SPARE", signal04 := "SBK3"."X1-2 GATE EC STACK 1 NG BOX PB.UNLOCK", signal05 := "SBK3"."X2-2 SPARE", signal06 := "SBK3"."X3-2 SPARE", signal07 := "SBK3"."X4-2 SPARE", signal08 :=, signal09 :=, signal10 :=, signal11 :=, signal12 :=, signal13 :=, signal14 :=, signal15 :=, interfaceSignals := "InstInterfaceSignals".statInterfaceSignalsHmi[40].valueSymbolLeft)
   END_RUNG
   // the same network as SCL:
   #instSignals40Left(signal00 := "SBK3"."X1-1 GATE EC STACK 1 NG BOX PB.LOCK",   // "LAF_InterfaceSignalsBool"
                      signal01 := "SBK3"."X2-1 GATE EC STACK 1 NG BOX PB.RESET",
                      signal02 := "SBK3"."X3-1 SPARE",
                      signal03 := "SBK3"."X4-1 SPARE",
                      signal04 := "SBK3"."X1-2 GATE EC STACK 1 NG BOX PB.UNLOCK",
                      signal05 := "SBK3"."X2-2 SPARE",
                      signal06 := "SBK3"."X3-2 SPARE",
                      signal07 := "SBK3"."X4-2 SPARE",
                      interfaceSignals := "InstInterfaceSignals".statInterfaceSignalsHmi[40].valueSymbolLeft);
END_REGION

REGION Network 46: Interface Signals 41 SBK04
   RUNG wire#powerrail
      #instSignals41Left(signal00 := "SBK4"."X1-1 GATE EC STACK 2 NG BOX PB.LOCK", signal01 := "SBK4"."X2-1 GATE EC STACK 2 NG BOX PB.RESET", signal02 := "SBK4"."X3-1 DIFFERENTIAL PRESSURE SWITCH NC", signal03 := "SBK4"."X4-1 DIFFERENTIAL PRESSURE SWITCH 2 NC", signal04 := "SBK4"."X1-2 GATE EC STACK 2 NG BOX PB.UNLOCK", signal05 := "SBK4"."X2-2 SPARE", signal06 := "SBK4"."X3-2 DIFFERENTIAL PRESSURE SWITCH NO", signal07 := "SBK4"."X4-2 DIFFERENTIAL PRESSURE SWITCH 2 NO", signal08 :=, signal09 :=, signal10 :=, signal11 :=, signal12 :=, signal13 :=, signal14 :=, signal15 :=, interfaceSignals := "InstInterfaceSignals".statInterfaceSignalsHmi[41].valueSymbolLeft)
   END_RUNG
   // the same network as SCL:
   #instSignals41Left(signal00 := "SBK4"."X1-1 GATE EC STACK 2 NG BOX PB.LOCK",   // "LAF_InterfaceSignalsBool"
                      signal01 := "SBK4"."X2-1 GATE EC STACK 2 NG BOX PB.RESET",
                      signal02 := "SBK4"."X3-1 DIFFERENTIAL PRESSURE SWITCH NC",
                      signal03 := "SBK4"."X4-1 DIFFERENTIAL PRESSURE SWITCH 2 NC",
                      signal04 := "SBK4"."X1-2 GATE EC STACK 2 NG BOX PB.UNLOCK",
                      signal05 := "SBK4"."X2-2 SPARE",
                      signal06 := "SBK4"."X3-2 DIFFERENTIAL PRESSURE SWITCH NO",
                      signal07 := "SBK4"."X4-2 DIFFERENTIAL PRESSURE SWITCH 2 NO",
                      interfaceSignals := "InstInterfaceSignals".statInterfaceSignalsHmi[41].valueSymbolLeft);
END_REGION

REGION Network 47: Interface Signals 42 SBK05
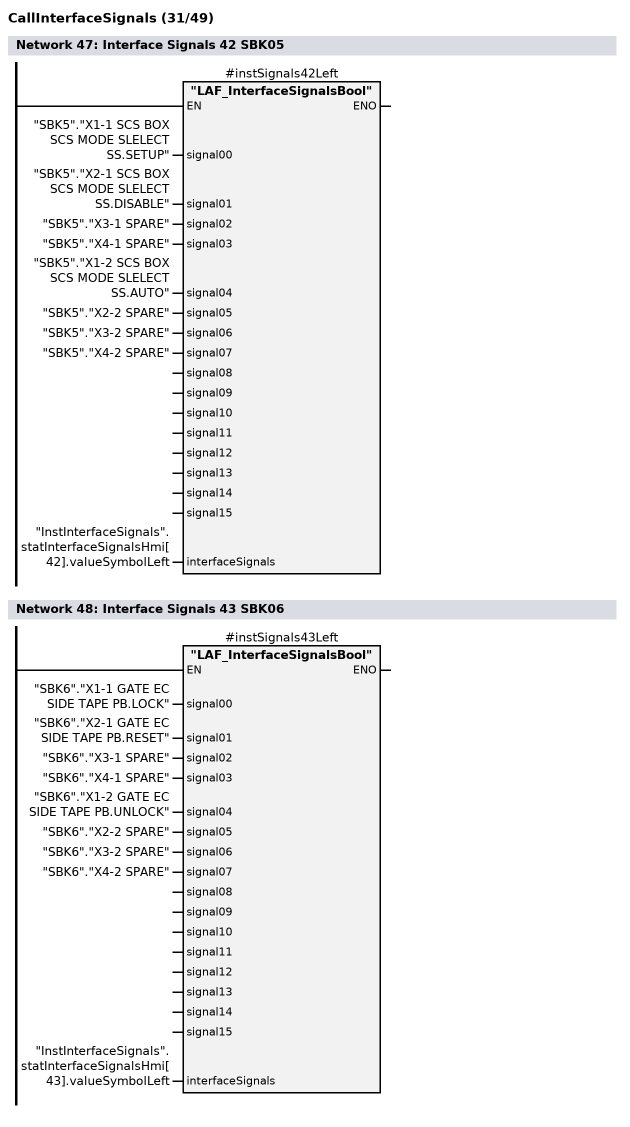
   RUNG wire#powerrail
      #instSignals42Left(signal00 := "SBK5"."X1-1 SCS BOX SCS MODE SLELECT SS.SETUP", signal01 := "SBK5"."X2-1 SCS BOX SCS MODE SLELECT SS.DISABLE", signal02 := "SBK5"."X3-1 SPARE", signal03 := "SBK5"."X4-1 SPARE", signal04 := "SBK5"."X1-2 SCS BOX SCS MODE SLELECT SS.AUTO", signal05 := "SBK5"."X2-2 SPARE", signal06 := "SBK5"."X3-2 SPARE", signal07 := "SBK5"."X4-2 SPARE", signal08 :=, signal09 :=, signal10 :=, signal11 :=, signal12 :=, signal13 :=, signal14 :=, signal15 :=, interfaceSignals := "InstInterfaceSignals".statInterfaceSignalsHmi[42].valueSymbolLeft)
   END_RUNG
   // the same network as SCL:
   #instSignals42Left(signal00 := "SBK5"."X1-1 SCS BOX SCS MODE SLELECT SS.SETUP",   // "LAF_InterfaceSignalsBool"
                      signal01 := "SBK5"."X2-1 SCS BOX SCS MODE SLELECT SS.DISABLE",
                      signal02 := "SBK5"."X3-1 SPARE",
                      signal03 := "SBK5"."X4-1 SPARE",
                      signal04 := "SBK5"."X1-2 SCS BOX SCS MODE SLELECT SS.AUTO",
                      signal05 := "SBK5"."X2-2 SPARE",
                      signal06 := "SBK5"."X3-2 SPARE",
                      signal07 := "SBK5"."X4-2 SPARE",
                      interfaceSignals := "InstInterfaceSignals".statInterfaceSignalsHmi[42].valueSymbolLeft);
END_REGION

REGION Network 48: Interface Signals 43 SBK06
   RUNG wire#powerrail
      #instSignals43Left(signal00 := "SBK6"."X1-1 GATE EC SIDE TAPE PB.LOCK", signal01 := "SBK6"."X2-1 GATE EC SIDE TAPE PB.RESET", signal02 := "SBK6"."X3-1 SPARE", signal03 := "SBK6"."X4-1 SPARE", signal04 := "SBK6"."X1-2 GATE EC SIDE TAPE PB.UNLOCK", signal05 := "SBK6"."X2-2 SPARE", signal06 := "SBK6"."X3-2 SPARE", signal07 := "SBK6"."X4-2 SPARE", signal08 :=, signal09 :=, signal10 :=, signal11 :=, signal12 :=, signal13 :=, signal14 :=, signal15 :=, interfaceSignals := "InstInterfaceSignals".statInterfaceSignalsHmi[43].valueSymbolLeft)
   END_RUNG
   // the same network as SCL:
   #instSignals43Left(signal00 := "SBK6"."X1-1 GATE EC SIDE TAPE PB.LOCK",   // "LAF_InterfaceSignalsBool"
                      signal01 := "SBK6"."X2-1 GATE EC SIDE TAPE PB.RESET",
                      signal02 := "SBK6"."X3-1 SPARE",
                      signal03 := "SBK6"."X4-1 SPARE",
                      signal04 := "SBK6"."X1-2 GATE EC SIDE TAPE PB.UNLOCK",
                      signal05 := "SBK6"."X2-2 SPARE",
                      signal06 := "SBK6"."X3-2 SPARE",
                      signal07 := "SBK6"."X4-2 SPARE",
                      interfaceSignals := "InstInterfaceSignals".statInterfaceSignalsHmi[43].valueSymbolLeft);
END_REGION

REGION Network 49: Interface Signals 44 SBK07
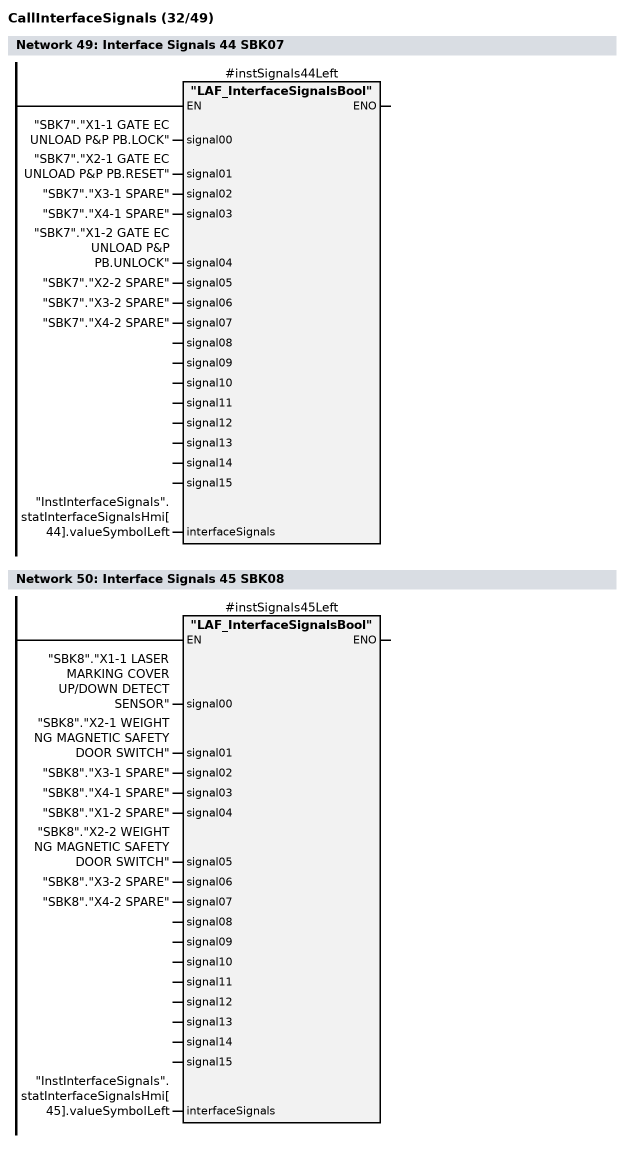
   RUNG wire#powerrail
      #instSignals44Left(signal00 := "SBK7"."X1-1 GATE EC UNLOAD P&P PB.LOCK", signal01 := "SBK7"."X2-1 GATE EC UNLOAD P&P PB.RESET", signal02 := "SBK7"."X3-1 SPARE", signal03 := "SBK7"."X4-1 SPARE", signal04 := "SBK7"."X1-2 GATE EC UNLOAD P&P PB.UNLOCK", signal05 := "SBK7"."X2-2 SPARE", signal06 := "SBK7"."X3-2 SPARE", signal07 := "SBK7"."X4-2 SPARE", signal08 :=, signal09 :=, signal10 :=, signal11 :=, signal12 :=, signal13 :=, signal14 :=, signal15 :=, interfaceSignals := "InstInterfaceSignals".statInterfaceSignalsHmi[44].valueSymbolLeft)
   END_RUNG
   // the same network as SCL:
   #instSignals44Left(signal00 := "SBK7"."X1-1 GATE EC UNLOAD P&P PB.LOCK",   // "LAF_InterfaceSignalsBool"
                      signal01 := "SBK7"."X2-1 GATE EC UNLOAD P&P PB.RESET",
                      signal02 := "SBK7"."X3-1 SPARE",
                      signal03 := "SBK7"."X4-1 SPARE",
                      signal04 := "SBK7"."X1-2 GATE EC UNLOAD P&P PB.UNLOCK",
                      signal05 := "SBK7"."X2-2 SPARE",
                      signal06 := "SBK7"."X3-2 SPARE",
                      signal07 := "SBK7"."X4-2 SPARE",
                      interfaceSignals := "InstInterfaceSignals".statInterfaceSignalsHmi[44].valueSymbolLeft);
END_REGION

REGION Network 50: Interface Signals 45 SBK08
   RUNG wire#powerrail
      #instSignals45Left(signal00 := "SBK8"."X1-1 LASER MARKING COVER UP/DOWN DETECT SENSOR", signal01 := "SBK8"."X2-1 WEIGHT NG MAGNETIC SAFETY DOOR SWITCH", signal02 := "SBK8"."X3-1 SPARE", signal03 := "SBK8"."X4-1 SPARE", signal04 := "SBK8"."X1-2 SPARE", signal05 := "SBK8"."X2-2 WEIGHT NG MAGNETIC SAFETY DOOR SWITCH", signal06 := "SBK8"."X3-2 SPARE", signal07 := "SBK8"."X4-2 SPARE", signal08 :=, signal09 :=, signal10 :=, signal11 :=, signal12 :=, signal13 :=, signal14 :=, signal15 :=, interfaceSignals := "InstInterfaceSignals".statInterfaceSignalsHmi[45].valueSymbolLeft)
   END_RUNG
   // the same network as SCL:
   #instSignals45Left(signal00 := "SBK8"."X1-1 LASER MARKING COVER UP/DOWN DETECT SENSOR",   // "LAF_InterfaceSignalsBool"
                      signal01 := "SBK8"."X2-1 WEIGHT NG MAGNETIC SAFETY DOOR SWITCH",
                      signal02 := "SBK8"."X3-1 SPARE",
                      signal03 := "SBK8"."X4-1 SPARE",
                      signal04 := "SBK8"."X1-2 SPARE",
                      signal05 := "SBK8"."X2-2 WEIGHT NG MAGNETIC SAFETY DOOR SWITCH",
                      signal06 := "SBK8"."X3-2 SPARE",
                      signal07 := "SBK8"."X4-2 SPARE",
                      interfaceSignals := "InstInterfaceSignals".statInterfaceSignalsHmi[45].valueSymbolLeft);
END_REGION

REGION Network 51: Interface Signals 46 SBK09
